LIN {X 0,Y 366.643,Z 618.897,A -85,B 0,C 180,E1 13820.841,E2 13820.841} C_VEL
LIN {X 0,Y 360.03,Z 667.651,A -85,B 0,C 180,E1 13819.206,E2 13819.206} C_VEL
LIN {X 0,Y 355.595,Z 700.826,A -85,B 0,C 180,E1 13817.811,E2 13817.811} C_VEL
LIN {X 0,Y 351.844,Z 722.205,A -85,B 0,C 180,E1 13816.612,E2 13816.612} C_VEL
LIN {X 0,Y 347.315,Z 742.561,A -85,B 0,C 180,E1 13815.174,E2 13815.174} C_VEL
LIN {X 0,Y 342.182,Z 761.879,A -85,B 0,C 180,E1 13813.484,E2 13813.484} C_VEL
LIN {X 0,Y 336.449,Z 780.451,A -85,B 0,C 180,E1 13811.503,E2 13811.503} C_VEL
LIN {X 0,Y 330.364,Z 797.932,A -85,B 0,C 180,E1 13809.24,E2 13809.24} C_VEL
LIN {X 0,Y 324.065,Z 814.382,A -85,B 0,C 180,E1 13806.657,E2 13806.657} C_VEL
LIN {X 0,Y 317.926,Z 829.258,A -85,B 0,C 180,E1 13803.826,E2 13803.826} C_VEL
LIN {X 0,Y 311.925,Z 843.014,A -85,B 0,C 180,E1 13800.643,E2 13800.643} C_VEL
LIN {X 0,Y 306.423,Z 855.219,A -85,B 0,C 180,E1 13797.183,E2 13797.183} C_VEL
LIN {X 0,Y 301.577,Z 865.858,A -85,B 0,C 180,E1 13793.445,E2 13793.445} C_VEL
LIN {X 0,Y 297.526,Z 874.902,A -85,B 0,C 180,E1 13789.433,E2 13789.433} C_VEL
LIN {X 0,Y 294.517,Z 881.994,A -85,B 0,C 180,E1 13785.356,E2 13785.356} C_VEL
LIN {X 0,Y 292.358,Z 887.482,A -85,B 0,C 180,E1 13781.042,E2 13781.042} C_VEL
LIN {X 0,Y 291.105,Z 891.11,A -85,B 0,C 180,E1 13776.707,E2 13776.707} C_VEL
LIN {X 0,Y 290.551,Z 892.885,A -85,B 0,C 180,E1 13772.564,E2 13772.564} C_VEL
LIN {X 0,Y 290.477,Z 893.097,A -85,B 0,C 180,E1 13768.619,E2 13768.619} C_VEL
LIN {X 0,Y 290.873,Z 891.794,A -85,B 0,C 180,E1 13764.477,E2 13764.477} C_VEL
LIN {X 0,Y 291.835,Z 888.902,A -85,B 0,C 180,E1 13760.335,E2 13760.335} C_VEL
LIN {X 0,Y 293.569,Z 884.354,A -85,B 0,C 180,E1 13756.207,E2 13756.207} C_VEL
LIN {X 0,Y 296.202,Z 878.044,A -85,B 0,C 180,E1 13752.11,E2 13752.11} C_VEL
LIN {X 0,Y 299.836,Z 869.83,A -85,B 0,C 180,E1 13748.069,E2 13748.069} C_VEL
LIN {X 0,Y 304.281,Z 860.081,A -85,B 0,C 180,E1 13744.294,E2 13744.294} C_VEL
LIN {X 0,Y 309.693,Z 848.18,A -85,B 0,C 180,E1 13740.61,E2 13740.61} C_VEL
LIN {X 0,Y 315.388,Z 835.383,A -85,B 0,C 180,E1 13737.387,E2 13737.387} C_VEL
LIN {X 0,Y 321.456,Z 821.111,A -85,B 0,C 180,E1 13734.432,E2 13734.432} C_VEL
LIN {X 0,Y 327.943,Z 804.743,A -85,B 0,C 180,E1 13731.65,E2 13731.65} C_VEL
LIN {X 0,Y 334.1,Z 787.79,A -85,B 0,C 180,E1 13729.275,E2 13729.275} C_VEL
LIN {X 0,Y 339.952,Z 769.852,A -85,B 0,C 180,E1 13727.201,E2 13727.201} C_VEL
LIN {X 0,Y 341.959,Z 763.048,A -85,B 0,C 180,E1 13726.517,E2 13726.517} C_VEL
LIN {X 0,Y 343.111,Z 756.729,A -85,B 0,C 180,E1 13725.787,E2 13725.787} C_VEL
LIN {X 0,Y 343.287,Z 740.949,A -85,B 0,C 180,E1 13723.705,E2 13723.705} C_VEL
LIN {X 0,Y 344.169,Z 734.277,A -85,B 0,C 180,E1 13723.068,E2 13723.068} C_VEL
LIN {X 0,Y 348.496,Z 713.392,A -85,B 0,C 180,E1 13721.732,E2 13721.732} C_VEL
LIN {X 0,Y 351.931,Z 691.641,A -85,B 0,C 180,E1 13720.649,E2 13720.649} C_VEL
LIN {X 0,Y 357.689,Z 649.532,A -85,B 0,C 180,E1 13719.026,E2 13719.026} C_VEL
LIN {X 0,Y 364.593,Z 600.879,A -85,B 0,C 180,E1 13717.565,E2 13717.565} C_VEL
LIN {X 0,Y 370.767,Z 550.378,A -85,B 0,C 180,E1 13716.308,E2 13716.308} C_VEL
LIN {X 0,Y 375.514,Z 499.907,A -85,B 0,C 180,E1 13715.262,E2 13715.262} C_VEL
LIN {X 0,Y 380.163,Z 439.411,A -85,B 0,C 180,E1 13714.164,E2 13714.164} C_VEL
LIN {X 0,Y 386.666,Z 411.148,A -85,B 0,C 180,E1 13713.223,E2 13713.223} C_VEL
LIN {X 0,Y 381.926,Z 396.352,A -85,B 0,C 180,E1 13710.437,E2 13710.437} C_VEL
LIN {X 0,Y 376.863,Z 382.161,A -85,B 0,C 180,E1 13707.323,E2 13707.323} C_VEL
LIN {X 0,Y 372.149,Z 370.419,A -85,B 0,C 180,E1 13704.273,E2 13704.273} C_VEL
LIN {X 0,Y 367.922,Z 360.719,A -85,B 0,C 180,E1 13701.315,E2 13701.315} C_VEL
LIN {X 0,Y 364.04,Z 352.331,A -85,B 0,C 180,E1 13698.247,E2 13698.247} C_VEL
LIN {X 0,Y 361.674,Z 347.588,A -85,B 0,C 180,E1 13696.214,E2 13696.214} C_VEL
LIN {X 0,Y 359.895,Z 343.923,A -85,B 0,C 180,E1 13694.48,E2 13694.48} C_VEL
LIN {X 0,Y 357.988,Z 339.875,A -85,B 0,C 180,E1 13692.256,E2 13692.256} C_VEL
LIN {X 0,Y 355.585,Z 335.237,A -85,B 0,C 180,E1 13689.223,E2 13689.223} C_VEL
LIN {X 0,Y 353.736,Z 331.636,A -85,B 0,C 180,E1 13685.841,E2 13685.841} C_VEL
LIN {X 0,Y 353.406,Z 330.304,A -85,B 0,C 180,E1 13684.706,E2 13684.706} C_VEL
LIN {X 0,Y 352.685,Z 328.775,A -85,B 0,C 180,E1 13678.375,E2 13678.375} C_VEL
LIN {X 0,Y 354.065,Z 329.807,A -85,B 0,C 180,E1 13673.677,E2 13673.677} C_VEL
LIN {X 0,Y 355.236,Z 330.811,A -85,B 0,C 180,E1 13671.828,E2 13671.828} C_VEL
LIN {X 0,Y 356.963,Z 342.871,A -85,B 0,C 180,E1 13667.626,E2 13667.626} C_VEL
LIN {X 0,Y 360.086,Z 356.086,A -85,B 0,C 180,E1 13663.671,E2 13663.671} C_VEL
LIN {X 0,Y 366.35,Z 375.856,A -85,B 0,C 180,E1 13658.715,E2 13658.715} C_VEL
LIN {X 0,Y 369.886,Z 385.971,A -85,B 0,C 180,E1 13656.543,E2 13656.543} C_VEL
LIN {X 0,Y 376.95,Z 407.665,A -85,B 0,C 180,E1 13652.729,E2 13652.729} C_VEL
LIN {X 0,Y 356.204,Z 579.083,A -85,B 0,C 180,E1 13648.165,E2 13648.165} C_VEL
LIN {X 0,Y 351.392,Z 648.87,A -85,B 0,C 180,E1 13646.675,E2 13646.675} C_VEL
LIN {X 0,Y 347.833,Z 683.011,A -85,B 0,C 180,E1 13645.721,E2 13645.721} C_VEL
LIN {X 0,Y 343.149,Z 716.181,A -85,B 0,C 180,E1 13644.541,E2 13644.541} C_VEL
LIN {X 0,Y 338.014,Z 746.973,A -85,B 0,C 180,E1 13643.133,E2 13643.133} C_VEL
LIN {X 0,Y 332.497,Z 776.814,A -85,B 0,C 180,E1 13641.433,E2 13641.433} C_VEL
LIN {X 0,Y 326.517,Z 805.796,A -85,B 0,C 180,E1 13639.415,E2 13639.415} C_VEL
LIN {X 0,Y 322.047,Z 824.838,A -85,B 0,C 180,E1 13637.773,E2 13637.773} C_VEL
LIN {X 0,Y 316.988,Z 843.135,A -85,B 0,C 180,E1 13635.845,E2 13635.845} C_VEL
LIN {X 0,Y 311.435,Z 861.14,A -85,B 0,C 180,E1 13633.525,E2 13633.525} C_VEL
LIN {X 0,Y 305.778,Z 878.186,A -85,B 0,C 180,E1 13630.844,E2 13630.844} C_VEL
LIN {X 0,Y 300.361,Z 893.477,A -85,B 0,C 180,E1 13627.911,E2 13627.911} C_VEL
LIN {X 0,Y 295.216,Z 907.713,A -85,B 0,C 180,E1 13624.61,E2 13624.61} C_VEL
LIN {X 0,Y 290.74,Z 920.364,A -85,B 0,C 180,E1 13621.055,E2 13621.055} C_VEL
LIN {X 0,Y 286.97,Z 931.798,A -85,B 0,C 180,E1 13617.158,E2 13617.158} C_VEL
LIN {X 0,Y 284.132,Z 941.659,A -85,B 0,C 180,E1 13612.993,E2 13612.993} C_VEL
LIN {X 0,Y 282.324,Z 949.983,A -85,B 0,C 180,E1 13608.587,E2 13608.587} C_VEL
LIN {X 0,Y 281.545,Z 956.442,A -85,B 0,C 180,E1 13604.176,E2 13604.176} C_VEL
LIN {X 0,Y 281.547,Z 960.921,A -85,B 0,C 180,E1 13600.021,E2 13600.021} C_VEL
LIN {X 0,Y 282.01,Z 964.446,A -85,B 0,C 180,E1 13595.289,E2 13595.289} C_VEL
LIN {X 0,Y 282.157,Z 966.76,A -85,B 0,C 180,E1 13591.624,E2 13591.624} C_VEL
LIN {X 0,Y 281.994,Z 967.796,A -85,B 0,C 180,E1 13588.171,E2 13588.171} C_VEL
LIN {X 0,Y 281.58,Z 967.758,A -85,B 0,C 180,E1 13584.702,E2 13584.702} C_VEL
LIN {X 0,Y 281.082,Z 966.455,A -85,B 0,C 180,E1 13580.582,E2 13580.582} C_VEL
LIN {X 0,Y 281.08,Z 963.184,A -85,B 0,C 180,E1 13575.581,E2 13575.581} C_VEL
LIN {X 0,Y 282.123,Z 958.691,A -85,B 0,C 180,E1 13570.97,E2 13570.97} C_VEL
LIN {X 0,Y 285.023,Z 951.705,A -85,B 0,C 180,E1 13565.546,E2 13565.546} C_VEL
LIN {X 0,Y 290.041,Z 942.875,A -85,B 0,C 180,E1 13560.236,E2 13560.236} C_VEL
LIN {X 0,Y 297.987,Z 931.43,A -85,B 0,C 180,E1 13554.75,E2 13554.75} C_VEL
LIN {X 0,Y 308.228,Z 918.66,A -85,B 0,C 180,E1 13549.792,E2 13549.792} C_VEL
LIN {X 0,Y 320.962,Z 904.077,A -85,B 0,C 180,E1 13545.246,E2 13545.246} C_VEL
LIN {X 0,Y 336.752,Z 887.173,A -85,B 0,C 180,E1 13541.011,E2 13541.011} C_VEL
LIN {X 0,Y 353.463,Z 870.171,A -85,B 0,C 180,E1 13537.62,E2 13537.62} C_VEL
LIN {X 0,Y 355.449,Z 868.133,A -85,B 0,C 180,E1 13537.244,E2 13537.244} C_VEL
LIN {X 0,Y 339.797,Z 879.829,A -85,B 0,C 180,E1 13534.197,E2 13534.197} C_VEL
LIN {X 0,Y 326.256,Z 889.867,A -85,B 0,C 180,E1 13530.785,E2 13530.785} C_VEL
LIN {X 0,Y 315.116,Z 897.821,A -85,B 0,C 180,E1 13527.189,E2 13527.189} C_VEL
LIN {X 0,Y 306.095,Z 903.73,A -85,B 0,C 180,E1 13523.486,E2 13523.486} C_VEL
LIN {X 0,Y 298.648,Z 907.843,A -85,B 0,C 180,E1 13519.561,E2 13519.561} C_VEL
LIN {X 0,Y 292.968,Z 909.937,A -85,B 0,C 180,E1 13515.642,E2 13515.642} C_VEL
LIN {X 0,Y 288.828,Z 910.181,A -85,B 0,C 180,E1 13511.786,E2 13511.786} C_VEL
LIN {X 0,Y 285.968,Z 908.753,A -85,B 0,C 180,E1 13508.04,E2 13508.04} C_VEL
LIN {X 0,Y 283.949,Z 905.358,A -85,B 0,C 180,E1 13504.039,E2 13504.039} C_VEL
LIN {X 0,Y 282.868,Z 900.293,A -85,B 0,C 180,E1 13500.203,E2 13500.203} C_VEL
LIN {X 0,Y 282.437,Z 893.734,A -85,B 0,C 180,E1 13496.55,E2 13496.55} C_VEL
LIN {X 0,Y 282.553,Z 885.362,A -85,B 0,C 180,E1 13492.885,E2 13492.885} C_VEL
LIN {X 0,Y 283.163,Z 875.563,A -85,B 0,C 180,E1 13489.419,E2 13489.419} C_VEL
LIN {X 0,Y 284.429,Z 862.976,A -85,B 0,C 180,E1 13485.754,E2 13485.754} C_VEL
LIN {X 0,Y 286.155,Z 849.601,A -85,B 0,C 180,E1 13482.512,E2 13482.512} C_VEL
LIN {X 0,Y 288.324,Z 834.796,A -85,B 0,C 180,E1 13479.496,E2 13479.496} C_VEL
LIN {X 0,Y 290.976,Z 818.009,A -85,B 0,C 180,E1 13476.605,E2 13476.605} C_VEL
LIN {X 0,Y 293.944,Z 799.899,A -85,B 0,C 180,E1 13473.972,E2 13473.972} C_VEL
LIN {X 0,Y 297.289,Z 779.355,A -85,B 0,C 180,E1 13471.471,E2 13471.471} C_VEL
LIN {X 0,Y 300.696,Z 757.667,A -85,B 0,C 180,E1 13469.308,E2 13469.308} C_VEL
LIN {X 0,Y 304.018,Z 734.908,A -85,B 0,C 180,E1 13467.47,E2 13467.47} C_VEL
LIN {X 0,Y 304.579,Z 731.096,A -85,B 0,C 180,E1 13467.184,E2 13467.184} C_VEL
LIN {X 0,Y 306.11,Z 730.891,A -85,B 0,C 180,E1 13466.718,E2 13466.718} C_VEL
LIN {X 0,Y 308.996,Z 728.323,A -85,B 0,C 180,E1 13466.18,E2 13466.18} C_VEL
LIN {X 0,Y 313.01,Z 722.831,A -85,B 0,C 180,E1 13465.68,E2 13465.68} C_VEL
LIN {X 0,Y 315.541,Z 718.67,A -85,B 0,C 180,E1 13465.443,E2 13465.443} C_VEL
LIN {X 0,Y 319.129,Z 715.537,A -85,B 0,C 180,E1 13464.795,E2 13464.795} C_VEL
LIN {X 0,Y 323.29,Z 709.874,A -85,B 0,C 180,E1 13464.256,E2 13464.256} C_VEL
LIN {X 0,Y 328.312,Z 700.656,A -85,B 0,C 180,E1 13463.823,E2 13463.823} C_VEL
LIN {X 0,Y 329.111,Z 699.455,A -85,B 0,C 180,E1 13463.723,E2 13463.723} C_VEL
LIN {X 0,Y 333.176,Z 694.404,A -85,B 0,C 180,E1 13463.141,E2 13463.141} C_VEL
LIN {X 0,Y 337.92,Z 686.155,A -85,B 0,C 180,E1 13462.657,E2 13462.657} C_VEL
LIN {X 0,Y 342.453,Z 676.446,A -85,B 0,C 180,E1 13462.34,E2 13462.34} C_VEL
LIN {X 0,Y 347.169,Z 669.599,A -85,B 0,C 180,E1 13461.766,E2 13461.766} C_VEL
LIN {X 0,Y 352.346,Z 659.543,A -85,B 0,C 180,E1 13461.329,E2 13461.329} C_VEL
LIN {X 0,Y 355.868,Z 651.493,A -85,B 0,C 180,E1 13461.105,E2 13461.105} C_VEL
LIN {X 0,Y 357.637,Z 649.135,A -85,B 0,C 180,E1 13460.884,E2 13460.884} C_VEL
LIN {X 0,Y 351.863,Z 690.96,A -85,B 0,C 180,E1 13459.267,E2 13459.267} C_VEL
LIN {X 0,Y 348.458,Z 712.778,A -85,B 0,C 180,E1 13458.189,E2 13458.189} C_VEL
LIN {X 0,Y 344.081,Z 734.017,A -85,B 0,C 180,E1 13456.836,E2 13456.836} C_VEL
LIN {X 0,Y 339.136,Z 753.596,A -85,B 0,C 180,E1 13455.28,E2 13455.28} C_VEL
LIN {X 0,Y 333.354,Z 772.976,A -85,B 0,C 180,E1 13453.384,E2 13453.384} C_VEL
LIN {X 0,Y 327.127,Z 791.223,A -85,B 0,C 180,E1 13451.2,E2 13451.2} C_VEL
LIN {X 0,Y 320.606,Z 808.342,A -85,B 0,C 180,E1 13448.705,E2 13448.705} C_VEL
LIN {X 0,Y 314.356,Z 823.41,A -85,B 0,C 180,E1 13446.047,E2 13446.047} C_VEL
LIN {X 0,Y 308.117,Z 837.495,A -85,B 0,C 180,E1 13443.038,E2 13443.038} C_VEL
LIN {X 0,Y 302.257,Z 850.138,A -85,B 0,C 180,E1 13439.75,E2 13439.75} C_VEL
LIN {X 0,Y 296.681,Z 861.846,A -85,B 0,C 180,E1 13435.985,E2 13435.985} C_VEL
LIN {X 0,Y 292.104,Z 871.467,A -85,B 0,C 180,E1 13432.12,E2 13432.12} C_VEL
LIN {X 0,Y 288.361,Z 879.551,A -85,B 0,C 180,E1 13427.975,E2 13427.975} C_VEL
LIN {X 0,Y 285.658,Z 885.743,A -85,B 0,C 180,E1 13423.77,E2 13423.77} C_VEL
LIN {X 0,Y 283.884,Z 890.175,A -85,B 0,C 180,E1 13419.524,E2 13419.524} C_VEL
LIN {X 0,Y 282.942,Z 892.841,A -85,B 0,C 180,E1 13415.475,E2 13415.475} C_VEL
LIN {X 0,Y 282.536,Z 894.107,A -85,B 0,C 180,E1 13411.217,E2 13411.217} C_VEL
LIN {X 0,Y 282.626,Z 893.861,A -85,B 0,C 180,E1 13407.161,E2 13407.161} C_VEL
LIN {X 0,Y 283.235,Z 892.063,A -85,B 0,C 180,E1 13402.903,E2 13402.903} C_VEL
LIN {X 0,Y 284.594,Z 888.422,A -85,B 0,C 180,E1 13398.448,E2 13398.448} C_VEL
LIN {X 0,Y 286.916,Z 882.914,A -85,B 0,C 180,E1 13394.02,E2 13394.02} C_VEL
LIN {X 0,Y 290.121,Z 875.798,A -85,B 0,C 180,E1 13389.84,E2 13389.84} C_VEL
LIN {X 0,Y 294.418,Z 866.728,A -85,B 0,C 180,E1 13385.736,E2 13385.736} C_VEL
LIN {X 0,Y 299.529,Z 856.058,A -85,B 0,C 180,E1 13381.921,E2 13381.921} C_VEL
LIN {X 0,Y 305.402,Z 843.624,A -85,B 0,C 180,E1 13378.348,E2 13378.348} C_VEL
LIN {X 0,Y 311.589,Z 830.016,A -85,B 0,C 180,E1 13375.166,E2 13375.166} C_VEL
LIN {X 0,Y 318.201,Z 814.584,A -85,B 0,C 180,E1 13372.211,E2 13372.211} C_VEL
LIN {X 0,Y 324.768,Z 797.965,A -85,B 0,C 180,E1 13369.603,E2 13369.603} C_VEL
LIN {X 0,Y 331.11,Z 780.235,A -85,B 0,C 180,E1 13367.317,E2 13367.317} C_VEL
LIN {X 0,Y 336.784,Z 762.36,A -85,B 0,C 180,E1 13365.412,E2 13365.412} C_VEL
LIN {X 0,Y 342.19,Z 742.493,A -85,B 0,C 180,E1 13363.681,E2 13363.681} C_VEL
LIN {X 0,Y 344.169,Z 734.277,A -85,B 0,C 180,E1 13363.068,E2 13363.068} C_VEL
LIN {X 0,Y 345.161,Z 727.504,A -85,B 0,C 180,E1 13362.456,E2 13362.456} C_VEL
LIN {X 0,Y 344.675,Z 710.571,A -85,B 0,C 180,E1 13360.65,E2 13360.65} C_VEL
LIN {X 0,Y 345.144,Z 703.415,A -85,B 0,C 180,E1 13360.16,E2 13360.16} C_VEL
LIN {X 0,Y 350.733,Z 664.574,A -85,B 0,C 180,E1 13358.521,E2 13358.521} C_VEL
LIN {X 0,Y 356.943,Z 622.303,A -85,B 0,C 180,E1 13357.123,E2 13357.123} C_VEL
LIN {X 0,Y 363.707,Z 572.194,A -85,B 0,C 180,E1 13355.791,E2 13355.791} C_VEL
LIN {X 0,Y 369.148,Z 521.87,A -85,B 0,C 180,E1 13354.67,E2 13354.67} C_VEL
LIN {X 0,Y 374.356,Z 456.234,A -85,B 0,C 180,E1 13353.457,E2 13353.457} C_VEL
LIN {X 0,Y 375.644,Z 442.026,A -85,B 0,C 180,E1 13353.187,E2 13353.187} C_VEL
LIN {X 0,Y 381.952,Z 414.888,A -85,B 0,C 180,E1 13352.305,E2 13352.305} C_VEL
LIN {X 0,Y 377.182,Z 399.775,A -85,B 0,C 180,E1 13349.369,E2 13349.369} C_VEL
LIN {X 0,Y 372.444,Z 386.352,A -85,B 0,C 180,E1 13346.294,E2 13346.294} C_VEL
LIN {X 0,Y 367.993,Z 374.96,A -85,B 0,C 180,E1 13343.203,E2 13343.203} C_VEL
LIN {X 0,Y 363.588,Z 364.648,A -85,B 0,C 180,E1 13339.897,E2 13339.897} C_VEL
LIN {X 0,Y 359.792,Z 356.235,A -85,B 0,C 180,E1 13336.55,E2 13336.55} C_VEL
LIN {X 0,Y 357.363,Z 351.267,A -85,B 0,C 180,E1 13334.171,E2 13334.171} C_VEL
LIN {X 0,Y 355.676,Z 347.381,A -85,B 0,C 180,E1 13332.007,E2 13332.007} C_VEL
LIN {X 0,Y 353.511,Z 342.934,A -85,B 0,C 180,E1 13329.114,E2 13329.114} C_VEL
LIN {X 0,Y 351.685,Z 339.321,A -85,B 0,C 180,E1 13325.675,E2 13325.675} C_VEL
LIN {X 0,Y 351.434,Z 338.035,A -85,B 0,C 180,E1 13324.569,E2 13324.569} C_VEL
LIN {X 0,Y 350.792,Z 336.546,A -85,B 0,C 180,E1 13318.203,E2 13318.203} C_VEL
LIN {X 0,Y 352.569,Z 337.811,A -85,B 0,C 180,E1 13313.159,E2 13313.159} C_VEL
LIN {X 0,Y 353.238,Z 338.552,A -85,B 0,C 180,E1 13312.068,E2 13312.068} C_VEL
LIN {X 0,Y 354.771,Z 350.186,A -85,B 0,C 180,E1 13308.044,E2 13308.044} C_VEL
LIN {X 0,Y 357.683,Z 362.885,A -85,B 0,C 180,E1 13304.225,E2 13304.225} C_VEL
LIN {X 0,Y 363.605,Z 382.359,A -85,B 0,C 180,E1 13299.307,E2 13299.307} C_VEL
LIN {X 0,Y 366.869,Z 392.296,A -85,B 0,C 180,E1 13297.146,E2 13297.146} C_VEL
LIN {X 0,Y 372.922,Z 411.537,A -85,B 0,C 180,E1 13293.732,E2 13293.732} C_VEL
LIN {X 0,Y 351.644,Z 581.817,A -85,B 0,C 180,E1 13289.192,E2 13289.192} C_VEL
LIN {X 0,Y 347.333,Z 643.921,A -85,B 0,C 180,E1 13287.885,E2 13287.885} C_VEL
LIN {X 0,Y 343.821,Z 677.097,A -85,B 0,C 180,E1 13286.978,E2 13286.978} C_VEL
LIN {X 0,Y 339.246,Z 709.541,A -85,B 0,C 180,E1 13285.859,E2 13285.859} C_VEL
LIN {X 0,Y 334.198,Z 739.62,A -85,B 0,C 180,E1 13284.561,E2 13284.561} C_VEL
LIN {X 0,Y 329.139,Z 766.452,A -85,B 0,C 180,E1 13283.092,E2 13283.092} C_VEL
LIN {X 0,Y 323.665,Z 792.898,A -85,B 0,C 180,E1 13281.388,E2 13281.388} C_VEL
LIN {X 0,Y 318.9,Z 813.963,A -85,B 0,C 180,E1 13279.767,E2 13279.767} C_VEL
LIN {X 0,Y 313.811,Z 833.029,A -85,B 0,C 180,E1 13277.936,E2 13277.936} C_VEL
LIN {X 0,Y 308.277,Z 851.263,A -85,B 0,C 180,E1 13275.785,E2 13275.785} C_VEL
LIN {X 0,Y 302.587,Z 868.119,A -85,B 0,C 180,E1 13273.366,E2 13273.366} C_VEL
LIN {X 0,Y 296.762,Z 884.18,A -85,B 0,C 180,E1 13270.563,E2 13270.563} C_VEL
LIN {X 0,Y 291.203,Z 898.921,A -85,B 0,C 180,E1 13267.427,E2 13267.427} C_VEL
LIN {X 0,Y 285.848,Z 912.994,A -85,B 0,C 180,E1 13263.792,E2 13263.792} C_VEL
LIN {X 0,Y 281.5,Z 924.876,A -85,B 0,C 180,E1 13260.055,E2 13260.055} C_VEL
LIN {X 0,Y 277.904,Z 935.632,A -85,B 0,C 180,E1 13255.908,E2 13255.908} C_VEL
LIN {X 0,Y 275.364,Z 944.751,A -85,B 0,C 180,E1 13251.515,E2 13251.515} C_VEL
LIN {X 0,Y 273.934,Z 952.193,A -85,B 0,C 180,E1 13246.978,E2 13246.978} C_VEL
LIN {X 0,Y 273.513,Z 957.825,A -85,B 0,C 180,E1 13242.456,E2 13242.456} C_VEL
LIN {X 0,Y 273.762,Z 961.703,A -85,B 0,C 180,E1 13237.978,E2 13237.978} C_VEL
LIN {X 0,Y 274.215,Z 964.141,A -85,B 0,C 180,E1 13233.763,E2 13233.763} C_VEL
LIN {X 0,Y 274.249,Z 965.886,A -85,B 0,C 180,E1 13230.418,E2 13230.418} C_VEL
LIN {X 0,Y 273.977,Z 966.635,A -85,B 0,C 180,E1 13227.071,E2 13227.071} C_VEL
LIN {X 0,Y 273.434,Z 966.354,A -85,B 0,C 180,E1 13223.28,E2 13223.28} C_VEL
LIN {X 0,Y 272.998,Z 964.568,A -85,B 0,C 180,E1 13218.593,E2 13218.593} C_VEL
LIN {X 0,Y 273.392,Z 961.021,A -85,B 0,C 180,E1 13213.643,E2 13213.643} C_VEL
LIN {X 0,Y 275.26,Z 955.619,A -85,B 0,C 180,E1 13208.252,E2 13208.252} C_VEL
LIN {X 0,Y 279.247,Z 948.099,A -85,B 0,C 180,E1 13202.721,E2 13202.721} C_VEL
LIN {X 0,Y 286.111,Z 938.203,A -85,B 0,C 180,E1 13196.963,E2 13196.963} C_VEL
LIN {X 0,Y 295.749,Z 926.427,A -85,B 0,C 180,E1 13191.532,E2 13191.532} C_VEL
LIN {X 0,Y 308.63,Z 912.329,A -85,B 0,C 180,E1 13186.364,E2 13186.364} C_VEL
LIN {X 0,Y 324.964,Z 895.932,A -85,B 0,C 180,E1 13181.609,E2 13181.609} C_VEL
LIN {X 0,Y 342.561,Z 879.263,A -85,B 0,C 180,E1 13177.804,E2 13177.804} C_VEL
LIN {X 0,Y 345.779,Z 876.2,A -85,B 0,C 180,E1 13177.183,E2 13177.183} C_VEL
LIN {X 0,Y 329.727,Z 887.067,A -85,B 0,C 180,E1 13173.916,E2 13173.916} C_VEL
LIN {X 0,Y 316.341,Z 895.907,A -85,B 0,C 180,E1 13170.38,E2 13170.38} C_VEL
LIN {X 0,Y 305.348,Z 902.734,A -85,B 0,C 180,E1 13166.655,E2 13166.655} C_VEL
LIN {X 0,Y 296.124,Z 907.761,A -85,B 0,C 180,E1 13162.64,E2 13162.64} C_VEL
LIN {X 0,Y 288.937,Z 910.728,A -85,B 0,C 180,E1 13158.565,E2 13158.565} C_VEL
LIN {X 0,Y 283.548,Z 911.729,A -85,B 0,C 180,E1 13154.5,E2 13154.5} C_VEL
LIN {X 0,Y 279.712,Z 910.927,A -85,B 0,C 180,E1 13150.504,E2 13150.504} C_VEL
LIN {X 0,Y 277.138,Z 908.494,A -85,B 0,C 180,E1 13146.63,E2 13146.63} C_VEL
LIN {X 0,Y 275.432,Z 904.039,A -85,B 0,C 180,E1 13142.497,E2 13142.497} C_VEL
LIN {X 0,Y 274.615,Z 897.929,A -85,B 0,C 180,E1 13138.539,E2 13138.539} C_VEL
LIN {X 0,Y 274.433,Z 890.313,A -85,B 0,C 180,E1 13134.774,E2 13134.774} C_VEL
LIN {X 0,Y 274.82,Z 880.793,A -85,B 0,C 180,E1 13130.999,E2 13130.999} C_VEL
LIN {X 0,Y 275.674,Z 870.498,A -85,B 0,C 180,E1 13127.643,E2 13127.643} C_VEL
LIN {X 0,Y 277.198,Z 857.439,A -85,B 0,C 180,E1 13124.089,E2 13124.089} C_VEL
LIN {X 0,Y 279.257,Z 842.882,A -85,B 0,C 180,E1 13120.767,E2 13120.767} C_VEL
LIN {X 0,Y 281.877,Z 826.293,A -85,B 0,C 180,E1 13117.584,E2 13117.584} C_VEL
LIN {X 0,Y 284.925,Z 807.951,A -85,B 0,C 180,E1 13114.651,E2 13114.651} C_VEL
LIN {X 0,Y 288.304,Z 787.762,A -85,B 0,C 180,E1 13111.97,E2 13111.97} C_VEL
LIN {X 0,Y 291.752,Z 766.54,A -85,B 0,C 180,E1 13109.635,E2 13109.635} C_VEL
LIN {X 0,Y 294.859,Z 747.2,A -85,B 0,C 180,E1 13107.832,E2 13107.832} C_VEL
LIN {X 0,Y 296.39,Z 747.01,A -85,B 0,C 180,E1 13107.332,E2 13107.332} C_VEL
LIN {X 0,Y 299.207,Z 744.812,A -85,B 0,C 180,E1 13106.766,E2 13106.766} C_VEL
LIN {X 0,Y 303.035,Z 740.398,A -85,B 0,C 180,E1 13106.253,E2 13106.253} C_VEL
LIN {X 0,Y 304.712,Z 738.085,A -85,B 0,C 180,E1 13106.093,E2 13106.093} C_VEL
LIN {X 0,Y 308.153,Z 735.594,A -85,B 0,C 180,E1 13105.4,E2 13105.4} C_VEL
LIN {X 0,Y 312.287,Z 731.048,A -85,B 0,C 180,E1 13104.807,E2 13104.807} C_VEL
LIN {X 0,Y 317.192,Z 724.171,A -85,B 0,C 180,E1 13104.325,E2 13104.325} C_VEL
LIN {X 0,Y 321.621,Z 719.801,A -85,B 0,C 180,E1 13103.63,E2 13103.63} C_VEL
LIN {X 0,Y 326.394,Z 713.32,A -85,B 0,C 180,E1 13103.099,E2 13103.099} C_VEL
LIN {X 0,Y 331.706,Z 704.206,A -85,B 0,C 180,E1 13102.652,E2 13102.652} C_VEL
LIN {X 0,Y 336.52,Z 698.024,A -85,B 0,C 180,E1 13102.044,E2 13102.044} C_VEL
LIN {X 0,Y 341.759,Z 688.852,A -85,B 0,C 180,E1 13101.558,E2 13101.558} C_VEL
LIN {X 0,Y 345.773,Z 680.521,A -85,B 0,C 180,E1 13101.292,E2 13101.292} C_VEL
LIN {X 0,Y 348.925,Z 676.153,A -85,B 0,C 180,E1 13100.917,E2 13100.917} C_VEL
LIN {X 0,Y 344.608,Z 705.687,A -85,B 0,C 180,E1 13099.61,E2 13099.61} C_VEL
LIN {X 0,Y 340.76,Z 725.9,A -85,B 0,C 180,E1 13098.439,E2 13098.439} C_VEL
LIN {X 0,Y 335.873,Z 746.278,A -85,B 0,C 180,E1 13096.958,E2 13096.958} C_VEL
LIN {X 0,Y 330.387,Z 765.45,A -85,B 0,C 180,E1 13095.231,E2 13095.231} C_VEL
LIN {X 0,Y 324.254,Z 783.887,A -85,B 0,C 180,E1 13093.202,E2 13093.202} C_VEL
LIN {X 0,Y 317.754,Z 801.203,A -85,B 0,C 180,E1 13090.884,E2 13090.884} C_VEL
LIN {X 0,Y 311.233,Z 817.009,A -85,B 0,C 180,E1 13088.32,E2 13088.32} C_VEL
LIN {X 0,Y 304.434,Z 832.212,A -85,B 0,C 180,E1 13085.314,E2 13085.314} C_VEL
LIN {X 0,Y 297.971,Z 845.825,A -85,B 0,C 180,E1 13082.019,E2 13082.019} C_VEL
LIN {X 0,Y 292.018,Z 857.892,A -85,B 0,C 180,E1 13078.421,E2 13078.421} C_VEL
LIN {X 0,Y 286.751,Z 868.407,A -85,B 0,C 180,E1 13074.516,E2 13074.516} C_VEL
LIN {X 0,Y 282.514,Z 876.971,A -85,B 0,C 180,E1 13070.511,E2 13070.511} C_VEL
LIN {X 0,Y 279.162,Z 884.043,A -85,B 0,C 180,E1 13066.223,E2 13066.223} C_VEL
LIN {X 0,Y 276.738,Z 889.511,A -85,B 0,C 180,E1 13061.674,E2 13061.674} C_VEL
LIN {X 0,Y 275.316,Z 893.121,A -85,B 0,C 180,E1 13057.093,E2 13057.093} C_VEL
LIN {X 0,Y 274.688,Z 894.887,A -85,B 0,C 180,E1 13052.712,E2 13052.712} C_VEL
LIN {X 0,Y 274.606,Z 895.099,A -85,B 0,C 180,E1 13048.54,E2 13048.54} C_VEL
LIN {X 0,Y 275.057,Z 893.802,A -85,B 0,C 180,E1 13044.158,E2 13044.158} C_VEL
LIN {X 0,Y 276.147,Z 890.921,A -85,B 0,C 180,E1 13039.78,E2 13039.78} C_VEL
LIN {X 0,Y 278.099,Z 886.385,A -85,B 0,C 180,E1 13035.423,E2 13035.423} C_VEL
LIN {X 0,Y 280.98,Z 880.228,A -85,B 0,C 180,E1 13031.189,E2 13031.189} C_VEL
LIN {X 0,Y 284.857,Z 872.344,A -85,B 0,C 180,E1 13027.069,E2 13027.069} C_VEL
LIN {X 0,Y 289.699,Z 862.703,A -85,B 0,C 180,E1 13023.119,E2 13023.119} C_VEL
LIN {X 0,Y 295.568,Z 850.942,A -85,B 0,C 180,E1 13019.281,E2 13019.281} C_VEL
LIN {X 0,Y 301.712,Z 838.27,A -85,B 0,C 180,E1 13015.939,E2 13015.939} C_VEL
LIN {X 0,Y 308.232,Z 824.136,A -85,B 0,C 180,E1 13012.888,E2 13012.888} C_VEL
LIN {X 0,Y 315.125,Z 808.088,A -85,B 0,C 180,E1 13010.05,E2 13010.05} C_VEL
LIN {X 0,Y 321.753,Z 791.181,A -85,B 0,C 180,E1 13007.596,E2 13007.596} C_VEL
LIN {X 0,Y 327.984,Z 773.454,A -85,B 0,C 180,E1 13005.479,E2 13005.479} C_VEL
LIN {X 0,Y 333.963,Z 753.88,A -85,B 0,C 180,E1 13003.569,E2 13003.569} C_VEL
LIN {X 0,Y 339.078,Z 734.096,A -85,B 0,C 180,E1 13002.003,E2 13002.003} C_VEL
LIN {X 0,Y 343.327,Z 713.93,A -85,B 0,C 180,E1 13000.721,E2 13000.721} C_VEL
LIN {X 0,Y 345.144,Z 703.415,A -85,B 0,C 180,E1 13000.16,E2 13000.16} C_VEL
LIN {X 0,Y 345.652,Z 696.184,A -85,B 0,C 180,E1 12999.693,E2 12999.693} C_VEL
LIN {X 0,Y 344.547,Z 678.435,A -85,B 0,C 180,E1 12998.131,E2 12998.131} C_VEL
LIN {X 0,Y 345.016,Z 671.14,A -85,B 0,C 180,E1 12997.707,E2 12997.707} C_VEL
LIN {X 0,Y 351.317,Z 629.328,A -85,B 0,C 180,E1 12996.269,E2 12996.269} C_VEL
LIN {X 0,Y 358.541,Z 578.262,A -85,B 0,C 180,E1 12994.878,E2 12994.878} C_VEL
LIN {X 0,Y 364.196,Z 528.171,A -85,B 0,C 180,E1 12993.748,E2 12993.748} C_VEL
LIN {X 0,Y 369.295,Z 466.763,A -85,B 0,C 180,E1 12992.597,E2 12992.597} C_VEL
LIN {X 0,Y 371.189,Z 444.83,A -85,B 0,C 180,E1 12992.193,E2 12992.193} C_VEL
LIN {X 0,Y 377.281,Z 418.51,A -85,B 0,C 180,E1 12991.34,E2 12991.34} C_VEL
LIN {X 0,Y 372.706,Z 403.689,A -85,B 0,C 180,E1 12988.35,E2 12988.35} C_VEL
LIN {X 0,Y 368.179,Z 390.746,A -85,B 0,C 180,E1 12985.277,E2 12985.277} C_VEL
LIN {X 0,Y 364.132,Z 380.11,A -85,B 0,C 180,E1 12982.268,E2 12982.268} C_VEL
LIN {X 0,Y 360.372,Z 371.096,A -85,B 0,C 180,E1 12979.28,E2 12979.28} C_VEL
LIN {X 0,Y 357.05,Z 363.402,A -85,B 0,C 180,E1 12976.179,E2 12976.179} C_VEL
LIN {X 0,Y 354.771,Z 358.473,A -85,B 0,C 180,E1 12973.778,E2 12973.778} C_VEL
LIN {X 0,Y 353.222,Z 354.758,A -85,B 0,C 180,E1 12971.677,E2 12971.677} C_VEL
LIN {X 0,Y 351.316,Z 350.5,A -85,B 0,C 180,E1 12968.841,E2 12968.841} C_VEL
LIN {X 0,Y 349.637,Z 346.785,A -85,B 0,C 180,E1 12965.333,E2 12965.333} C_VEL
LIN {X 0,Y 349.523,Z 345.779,A -85,B 0,C 180,E1 12964.43,E2 12964.43} C_VEL
LIN {X 0,Y 348.875,Z 344.313,A -85,B 0,C 180,E1 12958.193,E2 12958.193} C_VEL
LIN {X 0,Y 350.785,Z 345.628,A -85,B 0,C 180,E1 12953.124,E2 12953.124} C_VEL
LIN {X 0,Y 351.232,Z 346.212,A -85,B 0,C 180,E1 12952.352,E2 12952.352} C_VEL
LIN {X 0,Y 352.621,Z 357.497,A -85,B 0,C 180,E1 12948.468,E2 12948.468} C_VEL
LIN {X 0,Y 355.325,Z 369.691,A -85,B 0,C 180,E1 12944.787,E2 12944.787} C_VEL
LIN {X 0,Y 360.791,Z 388.654,A -85,B 0,C 180,E1 12939.95,E2 12939.95} C_VEL
LIN {X 0,Y 363.902,Z 398.437,A -85,B 0,C 180,E1 12937.802,E2 12937.802} C_VEL
LIN {X 0,Y 368.896,Z 415.425,A -85,B 0,C 180,E1 12934.752,E2 12934.752} C_VEL
LIN {X 0,Y 347.702,Z 578.804,A -85,B 0,C 180,E1 12930.386,E2 12930.386} C_VEL
LIN {X 0,Y 343.26,Z 640.84,A -85,B 0,C 180,E1 12929.077,E2 12929.077} C_VEL
LIN {X 0,Y 339.632,Z 674.063,A -85,B 0,C 180,E1 12928.177,E2 12928.177} C_VEL
LIN {X 0,Y 334.92,Z 706.612,A -85,B 0,C 180,E1 12927.069,E2 12927.069} C_VEL
LIN {X 0,Y 329.773,Z 736.672,A -85,B 0,C 180,E1 12925.791,E2 12925.791} C_VEL
LIN {X 0,Y 324.267,Z 764.925,A -85,B 0,C 180,E1 12924.266,E2 12924.266} C_VEL
LIN {X 0,Y 318.05,Z 793.74,A -85,B 0,C 180,E1 12922.395,E2 12922.395} C_VEL
LIN {X 0,Y 313.326,Z 813.545,A -85,B 0,C 180,E1 12920.847,E2 12920.847} C_VEL
LIN {X 0,Y 308.022,Z 832.534,A -85,B 0,C 180,E1 12919.002,E2 12919.002} C_VEL
LIN {X 0,Y 302.499,Z 849.927,A -85,B 0,C 180,E1 12916.928,E2 12916.928} C_VEL
LIN {X 0,Y 296.599,Z 866.61,A -85,B 0,C 180,E1 12914.524,E2 12914.524} C_VEL
LIN {X 0,Y 290.406,Z 882.917,A -85,B 0,C 180,E1 12911.645,E2 12911.645} C_VEL
LIN {X 0,Y 284.535,Z 897.684,A -85,B 0,C 180,E1 12908.462,E2 12908.462} C_VEL
LIN {X 0,Y 278.87,Z 911.797,A -85,B 0,C 180,E1 12904.757,E2 12904.757} C_VEL
LIN {X 0,Y 274.014,Z 924.334,A -85,B 0,C 180,E1 12900.721,E2 12900.721} C_VEL
LIN {X 0,Y 270.15,Z 935.188,A -85,B 0,C 180,E1 12896.369,E2 12896.369} C_VEL
LIN {X 0,Y 267.426,Z 944.444,A -85,B 0,C 180,E1 12891.725,E2 12891.725} C_VEL
LIN {X 0,Y 265.952,Z 951.758,A -85,B 0,C 180,E1 12887.053,E2 12887.053} C_VEL
LIN {X 0,Y 265.54,Z 957.219,A -85,B 0,C 180,E1 12882.394,E2 12882.394} C_VEL
LIN {X 0,Y 265.804,Z 960.804,A -85,B 0,C 180,E1 12878.001,E2 12878.001} C_VEL
LIN {X 0,Y 266.299,Z 962.817,A -85,B 0,C 180,E1 12873.875,E2 12873.875} C_VEL
LIN {X 0,Y 266.367,Z 964.649,A -85,B 0,C 180,E1 12870,E2 12870} C_VEL
LIN {X 0,Y 266.018,Z 965.374,A -85,B 0,C 180,E1 12866.552,E2 12866.552} C_VEL
LIN {X 0,Y 265.461,Z 965.112,A -85,B 0,C 180,E1 12862.86,E2 12862.86} C_VEL
LIN {X 0,Y 265.046,Z 963.601,A -85,B 0,C 180,E1 12858.466,E2 12858.466} C_VEL
LIN {X 0,Y 265.547,Z 959.968,A -85,B 0,C 180,E1 12852.92,E2 12852.92} C_VEL
LIN {X 0,Y 267.446,Z 955.13,A -85,B 0,C 180,E1 12847.814,E2 12847.814} C_VEL
LIN {X 0,Y 272.085,Z 947.409,A -85,B 0,C 180,E1 12841.701,E2 12841.701} C_VEL
LIN {X 0,Y 279.501,Z 937.848,A -85,B 0,C 180,E1 12835.83,E2 12835.83} C_VEL
LIN {X 0,Y 289.909,Z 926.294,A -85,B 0,C 180,E1 12830.275,E2 12830.275} C_VEL
LIN {X 0,Y 304.431,Z 911.944,A -85,B 0,C 180,E1 12824.81,E2 12824.81} C_VEL
LIN {X 0,Y 321.084,Z 896.78,A -85,B 0,C 180,E1 12820.274,E2 12820.274} C_VEL
LIN {X 0,Y 335.98,Z 883.69,A -85,B 0,C 180,E1 12817.113,E2 12817.113} C_VEL
LIN {X 0,Y 320.197,Z 893.303,A -85,B 0,C 180,E1 12813.769,E2 12813.769} C_VEL
LIN {X 0,Y 306.371,Z 901.354,A -85,B 0,C 180,E1 12809.956,E2 12809.956} C_VEL
LIN {X 0,Y 295.108,Z 907.303,A -85,B 0,C 180,E1 12805.918,E2 12805.918} C_VEL
LIN {X 0,Y 286.494,Z 911.032,A -85,B 0,C 180,E1 12801.928,E2 12801.928} C_VEL
LIN {X 0,Y 279.523,Z 912.961,A -85,B 0,C 180,E1 12797.701,E2 12797.701} C_VEL
LIN {X 0,Y 274.597,Z 913.028,A -85,B 0,C 180,E1 12793.691,E2 12793.691} C_VEL
LIN {X 0,Y 270.967,Z 911.374,A -85,B 0,C 180,E1 12789.558,E2 12789.558} C_VEL
LIN {X 0,Y 268.494,Z 907.861,A -85,B 0,C 180,E1 12785.342,E2 12785.342} C_VEL
LIN {X 0,Y 267.113,Z 902.722,A -85,B 0,C 180,E1 12781.287,E2 12781.287} C_VEL
LIN {X 0,Y 266.496,Z 895.934,A -85,B 0,C 180,E1 12777.305,E2 12777.305} C_VEL
LIN {X 0,Y 266.5,Z 887.774,A -85,B 0,C 180,E1 12773.537,E2 12773.537} C_VEL
LIN {X 0,Y 267.095,Z 877.385,A -85,B 0,C 180,E1 12769.648,E2 12769.648} C_VEL
LIN {X 0,Y 268.276,Z 865.508,A -85,B 0,C 180,E1 12765.98,E2 12765.98} C_VEL
LIN {X 0,Y 270.015,Z 852.195,A -85,B 0,C 180,E1 12762.545,E2 12762.545} C_VEL
LIN {X 0,Y 272.488,Z 835.962,A -85,B 0,C 180,E1 12759.036,E2 12759.036} C_VEL
LIN {X 0,Y 275.487,Z 817.977,A -85,B 0,C 180,E1 12755.786,E2 12755.786} C_VEL
LIN {X 0,Y 278.801,Z 798.85,A -85,B 0,C 180,E1 12752.904,E2 12752.904} C_VEL
LIN {X 0,Y 282.236,Z 778.557,A -85,B 0,C 180,E1 12750.382,E2 12750.382} C_VEL
LIN {X 0,Y 285.146,Z 761.379,A -85,B 0,C 180,E1 12748.543,E2 12748.543} C_VEL
LIN {X 0,Y 286.729,Z 761.147,A -85,B 0,C 180,E1 12747.99,E2 12747.99} C_VEL
LIN {X 0,Y 289.74,Z 758.909,A -85,B 0,C 180,E1 12747.357,E2 12747.357} C_VEL
LIN {X 0,Y 294.315,Z 754.082,A -85,B 0,C 180,E1 12746.724,E2 12746.724} C_VEL
LIN {X 0,Y 297.283,Z 752.301,A -85,B 0,C 180,E1 12746.059,E2 12746.059} C_VEL
LIN {X 0,Y 301.725,Z 748.238,A -85,B 0,C 180,E1 12745.365,E2 12745.365} C_VEL
LIN {X 0,Y 305.43,Z 743.832,A -85,B 0,C 180,E1 12744.944,E2 12744.944} C_VEL
LIN {X 0,Y 309.582,Z 740.494,A -85,B 0,C 180,E1 12744.225,E2 12744.225} C_VEL
LIN {X 0,Y 314.388,Z 735.324,A -85,B 0,C 180,E1 12743.63,E2 12743.63} C_VEL
LIN {X 0,Y 318.866,Z 729.325,A -85,B 0,C 180,E1 12743.206,E2 12743.206} C_VEL
LIN {X 0,Y 324.23,Z 723.906,A -85,B 0,C 180,E1 12742.478,E2 12742.478} C_VEL
LIN {X 0,Y 329.942,Z 716.128,A -85,B 0,C 180,E1 12741.923,E2 12741.923} C_VEL
LIN {X 0,Y 334.161,Z 709.076,A -85,B 0,C 180,E1 12741.625,E2 12741.625} C_VEL
LIN {X 0,Y 339.511,Z 702.211,A -85,B 0,C 180,E1 12741.004,E2 12741.004} C_VEL
LIN {X 0,Y 340.39,Z 701.1,A -85,B 0,C 180,E1 12740.902,E2 12740.902} C_VEL
LIN {X 0,Y 336.602,Z 721.861,A -85,B 0,C 180,E1 12739.768,E2 12739.768} C_VEL
LIN {X 0,Y 331.63,Z 743.031,A -85,B 0,C 180,E1 12738.302,E2 12738.302} C_VEL
LIN {X 0,Y 326.08,Z 762.53,A -85,B 0,C 180,E1 12736.614,E2 12736.614} C_VEL
LIN {X 0,Y 319.86,Z 781.204,A -85,B 0,C 180,E1 12734.629,E2 12734.629} C_VEL
LIN {X 0,Y 313.009,Z 799.27,A -85,B 0,C 180,E1 12732.279,E2 12732.279} C_VEL
LIN {X 0,Y 305.9,Z 816.106,A -85,B 0,C 180,E1 12729.598,E2 12729.598} C_VEL
LIN {X 0,Y 298.762,Z 831.616,A -85,B 0,C 180,E1 12726.565,E2 12726.565} C_VEL
LIN {X 0,Y 291.947,Z 845.488,A -85,B 0,C 180,E1 12723.229,E2 12723.229} C_VEL
LIN {X 0,Y 285.632,Z 857.785,A -85,B 0,C 180,E1 12719.577,E2 12719.577} C_VEL
LIN {X 0,Y 280.009,Z 868.505,A -85,B 0,C 180,E1 12715.6,E2 12715.6} C_VEL
LIN {X 0,Y 275.246,Z 877.627,A -85,B 0,C 180,E1 12711.301,E2 12711.301} C_VEL
LIN {X 0,Y 271.595,Z 884.884,A -85,B 0,C 180,E1 12706.822,E2 12706.822} C_VEL
LIN {X 0,Y 268.992,Z 890.399,A -85,B 0,C 180,E1 12702.144,E2 12702.144} C_VEL
LIN {X 0,Y 267.473,Z 893.986,A -85,B 0,C 180,E1 12697.518,E2 12697.518} C_VEL
LIN {X 0,Y 266.772,Z 895.828,A -85,B 0,C 180,E1 12693.008,E2 12693.008} C_VEL
LIN {X 0,Y 266.662,Z 896.121,A -85,B 0,C 180,E1 12688.711,E2 12688.711} C_VEL
LIN {X 0,Y 267.113,Z 894.908,A -85,B 0,C 180,E1 12684.199,E2 12684.199} C_VEL
LIN {X 0,Y 268.239,Z 892.115,A -85,B 0,C 180,E1 12679.693,E2 12679.693} C_VEL
LIN {X 0,Y 270.266,Z 887.671,A -85,B 0,C 180,E1 12675.21,E2 12675.21} C_VEL
LIN {X 0,Y 273.328,Z 881.472,A -85,B 0,C 180,E1 12670.778,E2 12670.778} C_VEL
LIN {X 0,Y 277.515,Z 873.376,A -85,B 0,C 180,E1 12666.426,E2 12666.426} C_VEL
LIN {X 0,Y 282.598,Z 863.747,A -85,B 0,C 180,E1 12662.387,E2 12662.387} C_VEL
LIN {X 0,Y 288.734,Z 851.984,A -85,B 0,C 180,E1 12658.472,E2 12658.472} C_VEL
LIN {X 0,Y 295.141,Z 839.32,A -85,B 0,C 180,E1 12655.071,E2 12655.071} C_VEL
LIN {X 0,Y 301.919,Z 825.203,A -85,B 0,C 180,E1 12651.976,E2 12651.976} C_VEL
LIN {X 0,Y 308.9,Z 809.554,A -85,B 0,C 180,E1 12649.167,E2 12649.167} C_VEL
LIN {X 0,Y 315.928,Z 792.228,A -85,B 0,C 180,E1 12646.624,E2 12646.624} C_VEL
LIN {X 0,Y 322.368,Z 774.489,A -85,B 0,C 180,E1 12644.489,E2 12644.489} C_VEL
LIN {X 0,Y 328.282,Z 755.819,A -85,B 0,C 180,E1 12642.645,E2 12642.645} C_VEL
LIN {X 0,Y 333.552,Z 736.201,A -85,B 0,C 180,E1 12641.069,E2 12641.069} C_VEL
LIN {X 0,Y 338.068,Z 715.486,A -85,B 0,C 180,E1 12639.737,E2 12639.737} C_VEL
LIN {X 0,Y 341.601,Z 694.386,A -85,B 0,C 180,E1 12638.675,E2 12638.675} C_VEL
LIN {X 0,Y 345.016,Z 671.14,A -85,B 0,C 180,E1 12637.707,E2 12637.707} C_VEL
LIN {X 0,Y 345.559,Z 663.804,A -85,B 0,C 180,E1 12637.291,E2 12637.291} C_VEL
LIN {X 0,Y 344.886,Z 645.737,A -85,B 0,C 180,E1 12635.826,E2 12635.826} C_VEL
LIN {X 0,Y 345.461,Z 638.348,A -85,B 0,C 180,E1 12635.453,E2 12635.453} C_VEL
LIN {X 0,Y 352.686,Z 589.505,A -85,B 0,C 180,E1 12634.08,E2 12634.08} C_VEL
LIN {X 0,Y 358.626,Z 541.142,A -85,B 0,C 180,E1 12632.942,E2 12632.942} C_VEL
LIN {X 0,Y 363.158,Z 492.249,A -85,B 0,C 180,E1 12631.98,E2 12631.98} C_VEL
LIN {X 0,Y 366.865,Z 447.449,A -85,B 0,C 180,E1 12631.172,E2 12631.172} C_VEL
LIN {X 0,Y 372.743,Z 422.289,A -85,B 0,C 180,E1 12630.375,E2 12630.375} C_VEL
LIN {X 0,Y 368.415,Z 408.009,A -85,B 0,C 180,E1 12627.389,E2 12627.389} C_VEL
LIN {X 0,Y 364.236,Z 395.66,A -85,B 0,C 180,E1 12624.36,E2 12624.36} C_VEL
LIN {X 0,Y 360.156,Z 384.746,A -85,B 0,C 180,E1 12621.157,E2 12621.157} C_VEL
LIN {X 0,Y 356.22,Z 374.962,A -85,B 0,C 180,E1 12617.689,E2 12617.689} C_VEL
LIN {X 0,Y 352.759,Z 366.756,A -85,B 0,C 180,E1 12614.025,E2 12614.025} C_VEL
LIN {X 0,Y 350.734,Z 362.044,A -85,B 0,C 180,E1 12611.278,E2 12611.278} C_VEL
LIN {X 0,Y 349.13,Z 358.063,A -85,B 0,C 180,E1 12608.565,E2 12608.565} C_VEL
LIN {X 0,Y 347.607,Z 354.308,A -85,B 0,C 180,E1 12605.033,E2 12605.033} C_VEL
LIN {X 0,Y 347.482,Z 353.459,A -85,B 0,C 180,E1 12604.125,E2 12604.125} C_VEL
LIN {X 0,Y 347.085,Z 352.111,A -85,B 0,C 180,E1 12598.184,E2 12598.184} C_VEL
LIN {X 0,Y 349.109,Z 353.469,A -85,B 0,C 180,E1 12593.091,E2 12593.091} C_VEL
LIN {X 0,Y 349.322,Z 353.983,A -85,B 0,C 180,E1 12592.641,E2 12592.641} C_VEL
LIN {X 0,Y 350.507,Z 364.551,A -85,B 0,C 180,E1 12588.981,E2 12588.981} C_VEL
LIN {X 0,Y 352.914,Z 376.48,A -85,B 0,C 180,E1 12585.353,E2 12585.353} C_VEL
LIN {X 0,Y 358.177,Z 395.672,A -85,B 0,C 180,E1 12580.428,E2 12580.428} C_VEL
LIN {X 0,Y 361.075,Z 404.965,A -85,B 0,C 180,E1 12578.389,E2 12578.389} C_VEL
LIN {X 0,Y 364.976,Z 419.19,A -85,B 0,C 180,E1 12575.794,E2 12575.794} C_VEL
LIN {X 0,Y 343.906,Z 575.914,A -85,B 0,C 180,E1 12571.605,E2 12571.605} C_VEL
LIN {X 0,Y 339.36,Z 637.568,A -85,B 0,C 180,E1 12570.3,E2 12570.3} C_VEL
LIN {X 0,Y 335.582,Z 671.204,A -85,B 0,C 180,E1 12569.4,E2 12569.4} C_VEL
LIN {X 0,Y 330.753,Z 703.669,A -85,B 0,C 180,E1 12568.31,E2 12568.31} C_VEL
LIN {X 0,Y 325.385,Z 734.286,A -85,B 0,C 180,E1 12567.025,E2 12567.025} C_VEL
LIN {X 0,Y 319.944,Z 761.293,A -85,B 0,C 180,E1 12565.594,E2 12565.594} C_VEL
LIN {X 0,Y 313.887,Z 788.844,A -85,B 0,C 180,E1 12563.855,E2 12563.855} C_VEL
LIN {X 0,Y 308.688,Z 810.28,A -85,B 0,C 180,E1 12562.219,E2 12562.219} C_VEL
LIN {X 0,Y 303.137,Z 829.589,A -85,B 0,C 180,E1 12560.371,E2 12560.371} C_VEL
LIN {X 0,Y 297.3,Z 847.226,A -85,B 0,C 180,E1 12558.3,E2 12558.3} C_VEL
LIN {X 0,Y 290.87,Z 864.744,A -85,B 0,C 180,E1 12555.786,E2 12555.786} C_VEL
LIN {X 0,Y 284.444,Z 880.988,A -85,B 0,C 180,E1 12552.911,E2 12552.911} C_VEL
LIN {X 0,Y 278.335,Z 895.629,A -85,B 0,C 180,E1 12549.75,E2 12549.75} C_VEL
LIN {X 0,Y 272.276,Z 909.882,A -85,B 0,C 180,E1 12545.985,E2 12545.985} C_VEL
LIN {X 0,Y 267.294,Z 921.921,A -85,B 0,C 180,E1 12542.086,E2 12542.086} C_VEL
LIN {X 0,Y 263.198,Z 932.582,A -85,B 0,C 180,E1 12537.858,E2 12537.858} C_VEL
LIN {X 0,Y 260.13,Z 941.834,A -85,B 0,C 180,E1 12533.267,E2 12533.267} C_VEL
LIN {X 0,Y 258.224,Z 949.726,A -85,B 0,C 180,E1 12528.279,E2 12528.279} C_VEL
LIN {X 0,Y 257.569,Z 955.485,A -85,B 0,C 180,E1 12523.469,E2 12523.469} C_VEL
LIN {X 0,Y 257.778,Z 959.51,A -85,B 0,C 180,E1 12518.701,E2 12518.701} C_VEL
LIN {X 0,Y 258.287,Z 961.671,A -85,B 0,C 180,E1 12514.44,E2 12514.44} C_VEL
LIN {X 0,Y 258.519,Z 962.811,A -85,B 0,C 180,E1 12511.108,E2 12511.108} C_VEL
LIN {X 0,Y 258.193,Z 964.018,A -85,B 0,C 180,E1 12507.114,E2 12507.114} C_VEL
LIN {X 0,Y 257.543,Z 963.94,A -85,B 0,C 180,E1 12502.863,E2 12502.863} C_VEL
LIN {X 0,Y 257.104,Z 962.669,A -85,B 0,C 180,E1 12498.534,E2 12498.534} C_VEL
LIN {X 0,Y 257.44,Z 959.909,A -85,B 0,C 180,E1 12493.529,E2 12493.529} C_VEL
LIN {X 0,Y 259.646,Z 954.661,A -85,B 0,C 180,E1 12487.35,E2 12487.35} C_VEL
LIN {X 0,Y 264.211,Z 947.807,A -85,B 0,C 180,E1 12481.401,E2 12481.401} C_VEL
LIN {X 0,Y 272.006,Z 938.514,A -85,B 0,C 180,E1 12475.265,E2 12475.265} C_VEL
LIN {X 0,Y 283.522,Z 926.959,A -85,B 0,C 180,E1 12469.274,E2 12469.274} C_VEL
LIN {X 0,Y 298.295,Z 913.641,A -85,B 0,C 180,E1 12463.889,E2 12463.889} C_VEL
LIN {X 0,Y 315.481,Z 899.188,A -85,B 0,C 180,E1 12459.337,E2 12459.337} C_VEL
LIN {X 0,Y 326.168,Z 890.562,A -85,B 0,C 180,E1 12457.052,E2 12457.052} C_VEL
LIN {X 0,Y 310.014,Z 899.337,A -85,B 0,C 180,E1 12453.472,E2 12453.472} C_VEL
LIN {X 0,Y 296.356,Z 906.225,A -85,B 0,C 180,E1 12449.512,E2 12449.512} C_VEL
LIN {X 0,Y 285.264,Z 911.069,A -85,B 0,C 180,E1 12445.317,E2 12445.317} C_VEL
LIN {X 0,Y 276.501,Z 913.864,A -85,B 0,C 180,E1 12440.978,E2 12440.978} C_VEL
LIN {X 0,Y 269.849,Z 914.678,A -85,B 0,C 180,E1 12436.578,E2 12436.578} C_VEL
LIN {X 0,Y 265.25,Z 913.719,A -85,B 0,C 180,E1 12432.408,E2 12432.408} C_VEL
LIN {X 0,Y 261.959,Z 911.019,A -85,B 0,C 180,E1 12428.119,E2 12428.119} C_VEL
LIN {X 0,Y 259.841,Z 906.46,A -85,B 0,C 180,E1 12423.751,E2 12423.751} C_VEL
LIN {X 0,Y 258.767,Z 900.288,A -85,B 0,C 180,E1 12419.557,E2 12419.557} C_VEL
LIN {X 0,Y 258.435,Z 892.664,A -85,B 0,C 180,E1 12415.562,E2 12415.562} C_VEL
LIN {X 0,Y 258.727,Z 883.15,A -85,B 0,C 180,E1 12411.555,E2 12411.555} C_VEL
LIN {X 0,Y 259.6,Z 872.174,A -85,B 0,C 180,E1 12407.77,E2 12407.77} C_VEL
LIN {X 0,Y 261.198,Z 858.773,A -85,B 0,C 180,E1 12403.916,E2 12403.916} C_VEL
LIN {X 0,Y 263.291,Z 844.477,A -85,B 0,C 180,E1 12400.476,E2 12400.476} C_VEL
LIN {X 0,Y 266.029,Z 827.779,A -85,B 0,C 180,E1 12397.107,E2 12397.107} C_VEL
LIN {X 0,Y 269.345,Z 808.814,A -85,B 0,C 180,E1 12393.902,E2 12393.902} C_VEL
LIN {X 0,Y 272.919,Z 788.641,A -85,B 0,C 180,E1 12391.079,E2 12391.079} C_VEL
LIN {X 0,Y 275.484,Z 774.071,A -85,B 0,C 180,E1 12389.309,E2 12389.309} C_VEL
LIN {X 0,Y 277.117,Z 773.825,A -85,B 0,C 180,E1 12388.696,E2 12388.696} C_VEL
LIN {X 0,Y 279.822,Z 772.019,A -85,B 0,C 180,E1 12388.072,E2 12388.072} C_VEL
LIN {X 0,Y 283.993,Z 768.125,A -85,B 0,C 180,E1 12387.405,E2 12387.405} C_VEL
LIN {X 0,Y 287.484,Z 766.13,A -85,B 0,C 180,E1 12386.589,E2 12386.589} C_VEL
LIN {X 0,Y 292.129,Z 762.099,A -85,B 0,C 180,E1 12385.852,E2 12385.852} C_VEL
LIN {X 0,Y 293.991,Z 760.179,A -85,B 0,C 180,E1 12385.627,E2 12385.627} C_VEL
LIN {X 0,Y 298.345,Z 757.201,A -85,B 0,C 180,E1 12384.798,E2 12384.798} C_VEL
LIN {X 0,Y 303.846,Z 751.934,A -85,B 0,C 180,E1 12384.051,E2 12384.051} C_VEL
LIN {X 0,Y 306.307,Z 749.242,A -85,B 0,C 180,E1 12383.783,E2 12383.783} C_VEL
LIN {X 0,Y 311.901,Z 744.537,A -85,B 0,C 180,E1 12382.963,E2 12382.963} C_VEL
LIN {X 0,Y 317.585,Z 738.191,A -85,B 0,C 180,E1 12382.353,E2 12382.353} C_VEL
LIN {X 0,Y 320.622,Z 734.323,A -85,B 0,C 180,E1 12382.094,E2 12382.094} C_VEL
LIN {X 0,Y 326.669,Z 728.199,A -85,B 0,C 180,E1 12381.36,E2 12381.36} C_VEL
LIN {X 0,Y 331.79,Z 721.533,A -85,B 0,C 180,E1 12380.9,E2 12380.9} C_VEL
LIN {X 0,Y 327.148,Z 741.267,A -85,B 0,C 180,E1 12379.556,E2 12379.556} C_VEL
LIN {X 0,Y 321.749,Z 760.218,A -85,B 0,C 180,E1 12377.965,E2 12377.965} C_VEL
LIN {X 0,Y 315.427,Z 779.078,A -85,B 0,C 180,E1 12376.02,E2 12376.02} C_VEL
LIN {X 0,Y 308.575,Z 796.943,A -85,B 0,C 180,E1 12373.761,E2 12373.761} C_VEL
LIN {X 0,Y 301.421,Z 813.63,A -85,B 0,C 180,E1 12371.184,E2 12371.184} C_VEL
LIN {X 0,Y 294.083,Z 829.245,A -85,B 0,C 180,E1 12368.229,E2 12368.229} C_VEL
LIN {X 0,Y 287.194,Z 842.907,A -85,B 0,C 180,E1 12365.062,E2 12365.062} C_VEL
LIN {X 0,Y 280.689,Z 855.168,A -85,B 0,C 180,E1 12361.578,E2 12361.578} C_VEL
LIN {X 0,Y 274.762,Z 866.016,A -85,B 0,C 180,E1 12357.763,E2 12357.763} C_VEL
LIN {X 0,Y 269.581,Z 875.414,A -85,B 0,C 180,E1 12353.614,E2 12353.614} C_VEL
LIN {X 0,Y 265.321,Z 883.278,A -85,B 0,C 180,E1 12349.14,E2 12349.14} C_VEL
LIN {X 0,Y 262.232,Z 889.286,A -85,B 0,C 180,E1 12344.576,E2 12344.576} C_VEL
LIN {X 0,Y 260.213,Z 893.564,A -85,B 0,C 180,E1 12339.958,E2 12339.958} C_VEL
LIN {X 0,Y 259.111,Z 896.158,A -85,B 0,C 180,E1 12335.314,E2 12335.314} C_VEL
LIN {X 0,Y 258.716,Z 897.151,A -85,B 0,C 180,E1 12330.886,E2 12330.886} C_VEL
LIN {X 0,Y 258.893,Z 896.681,A -85,B 0,C 180,E1 12326.236,E2 12326.236} C_VEL
LIN {X 0,Y 259.735,Z 894.645,A -85,B 0,C 180,E1 12321.588,E2 12321.588} C_VEL
LIN {X 0,Y 261.405,Z 891.002,A -85,B 0,C 180,E1 12316.957,E2 12316.957} C_VEL
LIN {X 0,Y 264.12,Z 885.658,A -85,B 0,C 180,E1 12312.371,E2 12312.371} C_VEL
LIN {X 0,Y 267.957,Z 878.492,A -85,B 0,C 180,E1 12307.859,E2 12307.859} C_VEL
LIN {X 0,Y 272.742,Z 869.847,A -85,B 0,C 180,E1 12303.667,E2 12303.667} C_VEL
LIN {X 0,Y 278.618,Z 859.197,A -85,B 0,C 180,E1 12299.601,E2 12299.601} C_VEL
LIN {X 0,Y 285.198,Z 846.976,A -85,B 0,C 180,E1 12295.878,E2 12295.878} C_VEL
LIN {X 0,Y 292.279,Z 833.18,A -85,B 0,C 180,E1 12292.487,E2 12292.487} C_VEL
LIN {X 0,Y 299.457,Z 818.252,A -85,B 0,C 180,E1 12289.501,E2 12289.501} C_VEL
LIN {X 0,Y 306.505,Z 802.316,A -85,B 0,C 180,E1 12286.887,E2 12286.887} C_VEL
LIN {X 0,Y 313.469,Z 784.852,A -85,B 0,C 180,E1 12284.541,E2 12284.541} C_VEL
LIN {X 0,Y 319.752,Z 767.032,A -85,B 0,C 180,E1 12282.572,E2 12282.572} C_VEL
LIN {X 0,Y 325.624,Z 747.606,A -85,B 0,C 180,E1 12280.82,E2 12280.82} C_VEL
LIN {X 0,Y 330.583,Z 728.05,A -85,B 0,C 180,E1 12279.395,E2 12279.395} C_VEL
LIN {X 0,Y 334.804,Z 706.92,A -85,B 0,C 180,E1 12278.17,E2 12278.17} C_VEL
LIN {X 0,Y 340.845,Z 668.017,A -85,B 0,C 180,E1 12276.488,E2 12276.488} C_VEL
LIN {X 0,Y 345.461,Z 638.348,A -85,B 0,C 180,E1 12275.453,E2 12275.453} C_VEL
LIN {X 0,Y 346.093,Z 630.92,A -85,B 0,C 180,E1 12275.092,E2 12275.092} C_VEL
LIN {X 0,Y 345.73,Z 611.532,A -85,B 0,C 180,E1 12273.656,E2 12273.656} C_VEL
LIN {X 0,Y 346.295,Z 605.133,A -85,B 0,C 180,E1 12273.369,E2 12273.369} C_VEL
LIN {X 0,Y 352.764,Z 556.34,A -85,B 0,C 180,E1 12272.17,E2 12272.17} C_VEL
LIN {X 0,Y 357.731,Z 508.112,A -85,B 0,C 180,E1 12271.178,E2 12271.178} C_VEL
LIN {X 0,Y 362.648,Z 450.247,A -85,B 0,C 180,E1 12270.129,E2 12270.129} C_VEL
LIN {X 0,Y 368.302,Z 426.072,A -85,B 0,C 180,E1 12269.37,E2 12269.37} C_VEL
LIN {X 0,Y 364.176,Z 412.156,A -85,B 0,C 180,E1 12266.366,E2 12266.366} C_VEL
LIN {X 0,Y 360.093,Z 399.779,A -85,B 0,C 180,E1 12263.179,E2 12263.179} C_VEL
LIN {X 0,Y 356.102,Z 388.919,A -85,B 0,C 180,E1 12259.819,E2 12259.819} C_VEL
LIN {X 0,Y 352.793,Z 380.573,A -85,B 0,C 180,E1 12256.634,E2 12256.634} C_VEL
LIN {X 0,Y 350.053,Z 373.712,A -85,B 0,C 180,E1 12253.462,E2 12253.462} C_VEL
LIN {X 0,Y 348.405,Z 369.611,A -85,B 0,C 180,E1 12251.086,E2 12251.086} C_VEL
LIN {X 0,Y 346.952,Z 365.624,A -85,B 0,C 180,E1 12248.285,E2 12248.285} C_VEL
LIN {X 0,Y 345.586,Z 361.831,A -85,B 0,C 180,E1 12244.73,E2 12244.73} C_VEL
LIN {X 0,Y 345.451,Z 361.14,A -85,B 0,C 180,E1 12243.817,E2 12243.817} C_VEL
LIN {X 0,Y 345.294,Z 359.908,A -85,B 0,C 180,E1 12238.175,E2 12238.175} C_VEL
LIN {X 0,Y 347.292,Z 361.192,A -85,B 0,C 180,E1 12233.359,E2 12233.359} C_VEL
LIN {X 0,Y 347.467,Z 361.736,A -85,B 0,C 180,E1 12232.934,E2 12232.934} C_VEL
LIN {X 0,Y 348.421,Z 371.605,A -85,B 0,C 180,E1 12229.5,E2 12229.5} C_VEL
LIN {X 0,Y 350.524,Z 383.357,A -85,B 0,C 180,E1 12225.899,E2 12225.899} C_VEL
LIN {X 0,Y 355.377,Z 401.98,A -85,B 0,C 180,E1 12221.079,E2 12221.079} C_VEL
LIN {X 0,Y 358.077,Z 411.08,A -85,B 0,C 180,E1 12219.058,E2 12219.058} C_VEL
LIN {X 0,Y 361.157,Z 423.112,A -85,B 0,C 180,E1 12216.855,E2 12216.855} C_VEL
LIN {X 0,Y 340.28,Z 572.859,A -85,B 0,C 180,E1 12212.853,E2 12212.853} C_VEL
LIN {X 0,Y 335.724,Z 633.339,A -85,B 0,C 180,E1 12211.575,E2 12211.575} C_VEL
LIN {X 0,Y 331.756,Z 667.831,A -85,B 0,C 180,E1 12210.666,E2 12210.666} C_VEL
LIN {X 0,Y 326.687,Z 701.265,A -85,B 0,C 180,E1 12209.56,E2 12209.56} C_VEL
LIN {X 0,Y 321.248,Z 731.396,A -85,B 0,C 180,E1 12208.32,E2 12208.32} C_VEL
LIN {X 0,Y 315.648,Z 758.328,A -85,B 0,C 180,E1 12206.915,E2 12206.915} C_VEL
LIN {X 0,Y 309.661,Z 785.042,A -85,B 0,C 180,E1 12205.263,E2 12205.263} C_VEL
LIN {X 0,Y 304.091,Z 807.531,A -85,B 0,C 180,E1 12203.576,E2 12203.576} C_VEL
LIN {X 0,Y 298.703,Z 825.778,A -85,B 0,C 180,E1 12201.873,E2 12201.873} C_VEL
LIN {X 0,Y 292.289,Z 844.528,A -85,B 0,C 180,E1 12199.717,E2 12199.717} C_VEL
LIN {X 0,Y 285.621,Z 862.049,A -85,B 0,C 180,E1 12197.223,E2 12197.223} C_VEL
LIN {X 0,Y 278.897,Z 878.424,A -85,B 0,C 180,E1 12194.355,E2 12194.355} C_VEL
LIN {X 0,Y 272.274,Z 893.536,A -85,B 0,C 180,E1 12191.098,E2 12191.098} C_VEL
LIN {X 0,Y 266.16,Z 907.221,A -85,B 0,C 180,E1 12187.487,E2 12187.487} C_VEL
LIN {X 0,Y 260.454,Z 920.133,A -85,B 0,C 180,E1 12183.297,E2 12183.297} C_VEL
LIN {X 0,Y 256.003,Z 930.92,A -85,B 0,C 180,E1 12178.967,E2 12178.967} C_VEL
LIN {X 0,Y 252.644,Z 940.22,A -85,B 0,C 180,E1 12174.305,E2 12174.305} C_VEL
LIN {X 0,Y 250.518,Z 947.999,A -85,B 0,C 180,E1 12169.346,E2 12169.346} C_VEL
LIN {X 0,Y 249.63,Z 954.104,A -85,B 0,C 180,E1 12164.226,E2 12164.226} C_VEL
LIN {X 0,Y 249.741,Z 958.149,A -85,B 0,C 180,E1 12159.448,E2 12159.448} C_VEL
LIN {X 0,Y 250.282,Z 960.475,A -85,B 0,C 180,E1 12155.042,E2 12155.042} C_VEL
LIN {X 0,Y 250.644,Z 961.382,A -85,B 0,C 180,E1 12151.143,E2 12151.143} C_VEL
LIN {X 0,Y 250.335,Z 962.567,A -85,B 0,C 180,E1 12147.253,E2 12147.253} C_VEL
LIN {X 0,Y 249.626,Z 962.76,A -85,B 0,C 180,E1 12142.867,E2 12142.867} C_VEL
LIN {X 0,Y 249.152,Z 961.367,A -85,B 0,C 180,E1 12137.719,E2 12137.719} C_VEL
LIN {X 0,Y 249.664,Z 958.616,A -85,B 0,C 180,E1 12132.52,E2 12132.52} C_VEL
LIN {X 0,Y 252.286,Z 953.52,A -85,B 0,C 180,E1 12126.155,E2 12126.155} C_VEL
LIN {X 0,Y 257.451,Z 946.724,A -85,B 0,C 180,E1 12120.008,E2 12120.008} C_VEL
LIN {X 0,Y 266.746,Z 937.029,A -85,B 0,C 180,E1 12113.338,E2 12113.338} C_VEL
LIN {X 0,Y 279.704,Z 925.495,A -85,B 0,C 180,E1 12107.217,E2 12107.217} C_VEL
LIN {X 0,Y 295.674,Z 912.532,A -85,B 0,C 180,E1 12101.928,E2 12101.928} C_VEL
LIN {X 0,Y 314.698,Z 898.105,A -85,B 0,C 180,E1 12097.363,E2 12097.363} C_VEL
LIN {X 0,Y 316.287,Z 896.898,A -85,B 0,C 180,E1 12096.99,E2 12096.99} C_VEL
LIN {X 0,Y 300.022,Z 904.665,A -85,B 0,C 180,E1 12093.226,E2 12093.226} C_VEL
LIN {X 0,Y 286.291,Z 910.541,A -85,B 0,C 180,E1 12089.043,E2 12089.043} C_VEL
LIN {X 0,Y 275.39,Z 914.302,A -85,B 0,C 180,E1 12084.68,E2 12084.68} C_VEL
LIN {X 0,Y 266.856,Z 916.048,A -85,B 0,C 180,E1 12080.165,E2 12080.165} C_VEL
LIN {X 0,Y 260.728,Z 915.908,A -85,B 0,C 180,E1 12075.8,E2 12075.8} C_VEL
LIN {X 0,Y 256.348,Z 914.113,A -85,B 0,C 180,E1 12071.474,E2 12071.474} C_VEL
LIN {X 0,Y 253.172,Z 910.306,A -85,B 0,C 180,E1 12066.805,E2 12066.805} C_VEL
LIN {X 0,Y 251.366,Z 904.758,A -85,B 0,C 180,E1 12062.28,E2 12062.28} C_VEL
LIN {X 0,Y 250.557,Z 897.616,A -85,B 0,C 180,E1 12057.942,E2 12057.942} C_VEL
LIN {X 0,Y 250.486,Z 889.011,A -85,B 0,C 180,E1 12053.813,E2 12053.813} C_VEL
LIN {X 0,Y 251.021,Z 879.044,A -85,B 0,C 180,E1 12049.906,E2 12049.906} C_VEL
LIN {X 0,Y 252.205,Z 867.049,A -85,B 0,C 180,E1 12046.005,E2 12046.005} C_VEL
LIN {X 0,Y 254.132,Z 852.773,A -85,B 0,C 180,E1 12042.128,E2 12042.128} C_VEL
LIN {X 0,Y 256.667,Z 836.908,A -85,B 0,C 180,E1 12038.519,E2 12038.519} C_VEL
LIN {X 0,Y 259.61,Z 820.001,A -85,B 0,C 180,E1 12035.298,E2 12035.298} C_VEL
LIN {X 0,Y 263.068,Z 800.909,A -85,B 0,C 180,E1 12032.25,E2 12032.25} C_VEL
LIN {X 0,Y 265.919,Z 785.589,A -85,B 0,C 180,E1 12030.118,E2 12030.118} C_VEL
LIN {X 0,Y 267.556,Z 785.32,A -85,B 0,C 180,E1 12029.453,E2 12029.453} C_VEL
LIN {X 0,Y 270.953,Z 783.098,A -85,B 0,C 180,E1 12028.645,E2 12028.645} C_VEL
LIN {X 0,Y 273.496,Z 780.839,A -85,B 0,C 180,E1 12028.233,E2 12028.233} C_VEL
LIN {X 0,Y 277.266,Z 778.882,A -85,B 0,C 180,E1 12027.252,E2 12027.252} C_VEL
LIN {X 0,Y 282.111,Z 774.981,A -85,B 0,C 180,E1 12026.433,E2 12026.433} C_VEL
LIN {X 0,Y 283.627,Z 773.906,A -85,B 0,C 180,E1 12026.151,E2 12026.151} C_VEL
LIN {X 0,Y 288,Z 771.06,A -85,B 0,C 180,E1 12025.293,E2 12025.293} C_VEL
LIN {X 0,Y 293.595,Z 766.149,A -85,B 0,C 180,E1 12024.514,E2 12024.514} C_VEL
LIN {X 0,Y 299.852,Z 761.546,A -85,B 0,C 180,E1 12023.48,E2 12023.48} C_VEL
LIN {X 0,Y 305.844,Z 755.879,A -85,B 0,C 180,E1 12022.784,E2 12022.784} C_VEL
LIN {X 0,Y 307.636,Z 754.215,A -85,B 0,C 180,E1 12022.57,E2 12022.57} C_VEL
LIN {X 0,Y 313.568,Z 749.089,A -85,B 0,C 180,E1 12021.784,E2 12021.784} C_VEL
LIN {X 0,Y 319.861,Z 742.293,A -85,B 0,C 180,E1 12021.188,E2 12021.188} C_VEL
LIN {X 0,Y 322.837,Z 738.833,A -85,B 0,C 180,E1 12020.929,E2 12020.929} C_VEL
LIN {X 0,Y 323.024,Z 738.715,A -85,B 0,C 180,E1 12020.899,E2 12020.899} C_VEL
LIN {X 0,Y 317.433,Z 758.321,A -85,B 0,C 180,E1 12019.305,E2 12019.305} C_VEL
LIN {X 0,Y 311.041,Z 777.243,A -85,B 0,C 180,E1 12017.405,E2 12017.405} C_VEL
LIN {X 0,Y 303.938,Z 795.536,A -85,B 0,C 180,E1 12015.15,E2 12015.15} C_VEL
LIN {X 0,Y 296.452,Z 812.676,A -85,B 0,C 180,E1 12012.552,E2 12012.552} C_VEL
LIN {X 0,Y 288.766,Z 828.6,A -85,B 0,C 180,E1 12009.578,E2 12009.578} C_VEL
LIN {X 0,Y 281.516,Z 842.523,A -85,B 0,C 180,E1 12006.381,E2 12006.381} C_VEL
LIN {X 0,Y 274.282,Z 855.624,A -85,B 0,C 180,E1 12002.652,E2 12002.652} C_VEL
LIN {X 0,Y 267.984,Z 866.636,A -85,B 0,C 180,E1 11998.738,E2 11998.738} C_VEL
LIN {X 0,Y 262.335,Z 876.359,A -85,B 0,C 180,E1 11994.363,E2 11994.363} C_VEL
LIN {X 0,Y 257.98,Z 883.994,A -85,B 0,C 180,E1 11989.943,E2 11989.943} C_VEL
LIN {X 0,Y 254.652,Z 890.073,A -85,B 0,C 180,E1 11985.253,E2 11985.253} C_VEL
LIN {X 0,Y 252.375,Z 894.573,A -85,B 0,C 180,E1 11980.27,E2 11980.27} C_VEL
LIN {X 0,Y 251.201,Z 897.161,A -85,B 0,C 180,E1 11975.482,E2 11975.482} C_VEL
LIN {X 0,Y 250.779,Z 898.152,A -85,B 0,C 180,E1 11970.914,E2 11970.914} C_VEL
LIN {X 0,Y 250.968,Z 897.684,A -85,B 0,C 180,E1 11966.117,E2 11966.117} C_VEL
LIN {X 0,Y 251.874,Z 895.635,A -85,B 0,C 180,E1 11961.298,E2 11961.298} C_VEL
LIN {X 0,Y 253.644,Z 892.014,A -85,B 0,C 180,E1 11956.551,E2 11956.551} C_VEL
LIN {X 0,Y 256.519,Z 886.679,A -85,B 0,C 180,E1 11951.83,E2 11951.83} C_VEL
LIN {X 0,Y 260.574,Z 879.522,A -85,B 0,C 180,E1 11947.197,E2 11947.197} C_VEL
LIN {X 0,Y 265.604,Z 870.883,A -85,B 0,C 180,E1 11942.902,E2 11942.902} C_VEL
LIN {X 0,Y 271.76,Z 860.242,A -85,B 0,C 180,E1 11938.749,E2 11938.749} C_VEL
LIN {X 0,Y 278.629,Z 848.026,A -85,B 0,C 180,E1 11934.958,E2 11934.958} C_VEL
LIN {X 0,Y 285.817,Z 834.602,A -85,B 0,C 180,E1 11931.595,E2 11931.595} C_VEL
LIN {X 0,Y 293.217,Z 819.817,A -85,B 0,C 180,E1 11928.582,E2 11928.582} C_VEL
LIN {X 0,Y 300.501,Z 803.968,A -85,B 0,C 180,E1 11925.939,E2 11925.939} C_VEL
LIN {X 0,Y 307.713,Z 786.538,A -85,B 0,C 180,E1 11923.563,E2 11923.563} C_VEL
LIN {X 0,Y 314.433,Z 768.065,A -85,B 0,C 180,E1 11921.506,E2 11921.506} C_VEL
LIN {X 0,Y 320.382,Z 749.009,A -85,B 0,C 180,E1 11919.777,E2 11919.777} C_VEL
LIN {X 0,Y 325.424,Z 729.786,A -85,B 0,C 180,E1 11918.365,E2 11918.365} C_VEL
LIN {X 0,Y 329.778,Z 708.764,A -85,B 0,C 180,E1 11917.134,E2 11917.134} C_VEL
LIN {X 0,Y 336.016,Z 670.139,A -85,B 0,C 180,E1 11915.443,E2 11915.443} C_VEL
LIN {X 0,Y 342.419,Z 630.14,A -85,B 0,C 180,E1 11914.076,E2 11914.076} C_VEL
LIN {X 0,Y 346.295,Z 605.133,A -85,B 0,C 180,E1 11913.369,E2 11913.369} C_VEL
LIN {X 0,Y 346.882,Z 597.672,A -85,B 0,C 180,E1 11913.024,E2 11913.024} C_VEL
LIN {X 0,Y 346.361,Z 578.132,A -85,B 0,C 180,E1 11911.648,E2 11911.648} C_VEL
LIN {X 0,Y 346.837,Z 571.682,A -85,B 0,C 180,E1 11911.387,E2 11911.387} C_VEL
LIN {X 0,Y 352.341,Z 523.727,A -85,B 0,C 180,E1 11910.353,E2 11910.353} C_VEL
LIN {X 0,Y 358.549,Z 453.065,A -85,B 0,C 180,E1 11909.063,E2 11909.063} C_VEL
LIN {X 0,Y 364.031,Z 430.052,A -85,B 0,C 180,E1 11908.371,E2 11908.371} C_VEL
LIN {X 0,Y 360.047,Z 416.391,A -85,B 0,C 180,E1 11905.32,E2 11905.32} C_VEL
LIN {X 0,Y 356.323,Z 404.78,A -85,B 0,C 180,E1 11902.204,E2 11902.204} C_VEL
LIN {X 0,Y 352.921,Z 395.214,A -85,B 0,C 180,E1 11899.144,E2 11899.144} C_VEL
LIN {X 0,Y 349.976,Z 387.363,A -85,B 0,C 180,E1 11896.089,E2 11896.089} C_VEL
LIN {X 0,Y 347.406,Z 380.655,A -85,B 0,C 180,E1 11892.889,E2 11892.889} C_VEL
LIN {X 0,Y 345.934,Z 376.873,A -85,B 0,C 180,E1 11890.66,E2 11890.66} C_VEL
LIN {X 0,Y 344.819,Z 373.303,A -85,B 0,C 180,E1 11888.169,E2 11888.169} C_VEL
LIN {X 0,Y 343.577,Z 369.463,A -85,B 0,C 180,E1 11884.507,E2 11884.507} C_VEL
LIN {X 0,Y 343.43,Z 368.82,A -85,B 0,C 180,E1 11883.505,E2 11883.505} C_VEL
LIN {X 0,Y 343.479,Z 367.699,A -85,B 0,C 180,E1 11878.332,E2 11878.332} C_VEL
LIN {X 0,Y 345.279,Z 368.86,A -85,B 0,C 180,E1 11873.682,E2 11873.682} C_VEL
LIN {X 0,Y 345.488,Z 369.332,A -85,B 0,C 180,E1 11873.269,E2 11873.269} C_VEL
LIN {X 0,Y 346.364,Z 378.658,A -85,B 0,C 180,E1 11870.026,E2 11870.026} C_VEL
LIN {X 0,Y 348.175,Z 390.05,A -85,B 0,C 180,E1 11866.506,E2 11866.506} C_VEL
LIN {X 0,Y 352.845,Z 408.971,A -85,B 0,C 180,E1 11861.581,E2 11861.581} C_VEL
LIN {X 0,Y 355.205,Z 417.496,A -85,B 0,C 180,E1 11859.678,E2 11859.678} C_VEL
LIN {X 0,Y 357.47,Z 426.949,A -85,B 0,C 180,E1 11857.939,E2 11857.939} C_VEL
LIN {X 0,Y 336.817,Z 569.861,A -85,B 0,C 180,E1 11854.126,E2 11854.126} C_VEL
LIN {X 0,Y 332.163,Z 629.931,A -85,B 0,C 180,E1 11852.855,E2 11852.855} C_VEL
LIN {X 0,Y 328.077,Z 664.549,A -85,B 0,C 180,E1 11851.958,E2 11851.958} C_VEL
LIN {X 0,Y 322.786,Z 698.857,A -85,B 0,C 180,E1 11850.839,E2 11850.839} C_VEL
LIN {X 0,Y 316.896,Z 730.284,A -85,B 0,C 180,E1 11849.561,E2 11849.561} C_VEL
LIN {X 0,Y 311.115,Z 757.419,A -85,B 0,C 180,E1 11848.161,E2 11848.161} C_VEL
LIN {X 0,Y 304.372,Z 786.191,A -85,B 0,C 180,E1 11846.363,E2 11846.363} C_VEL
LIN {X 0,Y 299.425,Z 805.619,A -85,B 0,C 180,E1 11844.9,E2 11844.9} C_VEL
LIN {X 0,Y 293.873,Z 823.687,A -85,B 0,C 180,E1 11843.236,E2 11843.236} C_VEL
LIN {X 0,Y 287.194,Z 842.545,A -85,B 0,C 180,E1 11841.082,E2 11841.082} C_VEL
LIN {X 0,Y 280.407,Z 859.77,A -85,B 0,C 180,E1 11838.643,E2 11838.643} C_VEL
LIN {X 0,Y 273.402,Z 876.134,A -85,B 0,C 180,E1 11835.792,E2 11835.792} C_VEL
LIN {X 0,Y 266.367,Z 891.442,A -85,B 0,C 180,E1 11832.507,E2 11832.507} C_VEL
LIN {X 0,Y 259.868,Z 905.271,A -85,B 0,C 180,E1 11828.842,E2 11828.842} C_VEL
LIN {X 0,Y 253.731,Z 918.322,A -85,B 0,C 180,E1 11824.574,E2 11824.574} C_VEL
LIN {X 0,Y 248.904,Z 929.249,A -85,B 0,C 180,E1 11820.142,E2 11820.142} C_VEL
LIN {X 0,Y 245.191,Z 938.697,A -85,B 0,C 180,E1 11815.353,E2 11815.353} C_VEL
LIN {X 0,Y 242.779,Z 946.583,A -85,B 0,C 180,E1 11810.24,E2 11810.24} C_VEL
LIN {X 0,Y 241.703,Z 952.882,A -85,B 0,C 180,E1 11804.861,E2 11804.861} C_VEL
LIN {X 0,Y 241.721,Z 956.944,A -85,B 0,C 180,E1 11800.005,E2 11800.005} C_VEL
LIN {X 0,Y 242.274,Z 959.368,A -85,B 0,C 180,E1 11795.447,E2 11795.447} C_VEL
LIN {X 0,Y 242.69,Z 960.344,A -85,B 0,C 180,E1 11791.416,E2 11791.416} C_VEL
LIN {X 0,Y 242.617,Z 960.808,A -85,B 0,C 180,E1 11788.347,E2 11788.347} C_VEL
LIN {X 0,Y 241.989,Z 961.423,A -85,B 0,C 180,E1 11784.309,E2 11784.309} C_VEL
LIN {X 0,Y 241.324,Z 960.912,A -85,B 0,C 180,E1 11779.737,E2 11779.737} C_VEL
LIN {X 0,Y 241.346,Z 959.091,A -85,B 0,C 180,E1 11774.624,E2 11774.624} C_VEL
LIN {X 0,Y 243.205,Z 954.97,A -85,B 0,C 180,E1 11768.029,E2 11768.029} C_VEL
LIN {X 0,Y 247.543,Z 949.265,A -85,B 0,C 180,E1 11761.71,E2 11761.71} C_VEL
LIN {X 0,Y 256.061,Z 940.692,A -85,B 0,C 180,E1 11754.695,E2 11754.695} C_VEL
LIN {X 0,Y 268.48,Z 930.238,A -85,B 0,C 180,E1 11748.191,E2 11748.191} C_VEL
LIN {X 0,Y 284.499,Z 918.06,A -85,B 0,C 180,E1 11742.434,E2 11742.434} C_VEL
LIN {X 0,Y 303.916,Z 904.379,A -85,B 0,C 180,E1 11737.492,E2 11737.492} C_VEL
LIN {X 0,Y 306.388,Z 902.677,A -85,B 0,C 180,E1 11736.938,E2 11736.938} C_VEL
LIN {X 0,Y 290.077,Z 909.42,A -85,B 0,C 180,E1 11732.999,E2 11732.999} C_VEL
LIN {X 0,Y 276.681,Z 914.167,A -85,B 0,C 180,E1 11728.728,E2 11728.728} C_VEL
LIN {X 0,Y 266.306,Z 916.874,A -85,B 0,C 180,E1 11724.394,E2 11724.394} C_VEL
LIN {X 0,Y 258.186,Z 917.772,A -85,B 0,C 180,E1 11719.926,E2 11719.926} C_VEL
LIN {X 0,Y 251.859,Z 916.837,A -85,B 0,C 180,E1 11715.19,E2 11715.19} C_VEL
LIN {X 0,Y 247.469,Z 914.048,A -85,B 0,C 180,E1 11710.476,E2 11710.476} C_VEL
LIN {X 0,Y 244.669,Z 909.579,A -85,B 0,C 180,E1 11705.864,E2 11705.864} C_VEL
LIN {X 0,Y 243.134,Z 903.597,A -85,B 0,C 180,E1 11701.414,E2 11701.414} C_VEL
LIN {X 0,Y 242.48,Z 895.781,A -85,B 0,C 180,E1 11696.927,E2 11696.927} C_VEL
LIN {X 0,Y 242.581,Z 886.484,A -85,B 0,C 180,E1 11692.659,E2 11692.659} C_VEL
LIN {X 0,Y 243.385,Z 875.099,A -85,B 0,C 180,E1 11688.387,E2 11688.387} C_VEL
LIN {X 0,Y 244.879,Z 862.174,A -85,B 0,C 180,E1 11684.366,E2 11684.366} C_VEL
LIN {X 0,Y 247.165,Z 846.76,A -85,B 0,C 180,E1 11680.38,E2 11680.38} C_VEL
LIN {X 0,Y 250.095,Z 829.651,A -85,B 0,C 180,E1 11676.684,E2 11676.684} C_VEL
LIN {X 0,Y 253.558,Z 810.82,A -85,B 0,C 180,E1 11673.285,E2 11673.285} C_VEL
LIN {X 0,Y 256.349,Z 796.184,A -85,B 0,C 180,E1 11671.015,E2 11671.015} C_VEL
LIN {X 0,Y 258.063,Z 795.879,A -85,B 0,C 180,E1 11670.267,E2 11670.267} C_VEL
LIN {X 0,Y 261.396,Z 793.79,A -85,B 0,C 180,E1 11669.419,E2 11669.419} C_VEL
LIN {X 0,Y 263.426,Z 792.151,A -85,B 0,C 180,E1 11669.048,E2 11669.048} C_VEL
LIN {X 0,Y 266.688,Z 790.708,A -85,B 0,C 180,E1 11668.085,E2 11668.085} C_VEL
LIN {X 0,Y 271.264,Z 787.43,A -85,B 0,C 180,E1 11667.19,E2 11667.19} C_VEL
LIN {X 0,Y 272.706,Z 786.509,A -85,B 0,C 180,E1 11666.885,E2 11666.885} C_VEL
LIN {X 0,Y 276.903,Z 784.082,A -85,B 0,C 180,E1 11665.965,E2 11665.965} C_VEL
LIN {X 0,Y 281.977,Z 780.134,A -85,B 0,C 180,E1 11665.186,E2 11665.186} C_VEL
LIN {X 0,Y 287.29,Z 776.786,A -85,B 0,C 180,E1 11664.188,E2 11664.188} C_VEL
LIN {X 0,Y 294.134,Z 771.195,A -85,B 0,C 180,E1 11663.251,E2 11663.251} C_VEL
LIN {X 0,Y 300.69,Z 766.466,A -85,B 0,C 180,E1 11662.276,E2 11662.276} C_VEL
LIN {X 0,Y 308.157,Z 759.605,A -85,B 0,C 180,E1 11661.465,E2 11661.465} C_VEL
LIN {X 0,Y 313.629,Z 755.169,A -85,B 0,C 180,E1 11660.78,E2 11660.78} C_VEL
LIN {X 0,Y 307.091,Z 774.598,A -85,B 0,C 180,E1 11658.904,E2 11658.904} C_VEL
LIN {X 0,Y 299.717,Z 793.413,A -85,B 0,C 180,E1 11656.659,E2 11656.659} C_VEL
LIN {X 0,Y 292.142,Z 810.488,A -85,B 0,C 180,E1 11654.147,E2 11654.147} C_VEL
LIN {X 0,Y 284.54,Z 825.999,A -85,B 0,C 180,E1 11651.349,E2 11651.349} C_VEL
LIN {X 0,Y 276.841,Z 840.469,A -85,B 0,C 180,E1 11648.142,E2 11648.142} C_VEL
LIN {X 0,Y 269.273,Z 853.798,A -85,B 0,C 180,E1 11644.477,E2 11644.477} C_VEL
LIN {X 0,Y 262.342,Z 865.452,A -85,B 0,C 180,E1 11640.459,E2 11640.459} C_VEL
LIN {X 0,Y 256.338,Z 875.316,A -85,B 0,C 180,E1 11636.154,E2 11636.154} C_VEL
LIN {X 0,Y 251.296,Z 883.626,A -85,B 0,C 180,E1 11631.473,E2 11631.473} C_VEL
LIN {X 0,Y 247.54,Z 890.026,A -85,B 0,C 180,E1 11626.666,E2 11626.666} C_VEL
LIN {X 0,Y 244.982,Z 894.672,A -85,B 0,C 180,E1 11621.775,E2 11621.775} C_VEL
LIN {X 0,Y 243.461,Z 897.762,A -85,B 0,C 180,E1 11616.604,E2 11616.604} C_VEL
LIN {X 0,Y 242.869,Z 899.092,A -85,B 0,C 180,E1 11611.652,E2 11611.652} C_VEL
LIN {X 0,Y 242.961,Z 898.929,A -85,B 0,C 180,E1 11606.933,E2 11606.933} C_VEL
LIN {X 0,Y 243.762,Z 897.219,A -85,B 0,C 180,E1 11601.983,E2 11601.983} C_VEL
LIN {X 0,Y 245.567,Z 893.689,A -85,B 0,C 180,E1 11596.82,E2 11596.82} C_VEL
LIN {X 0,Y 248.612,Z 888.313,A -85,B 0,C 180,E1 11591.717,E2 11591.717} C_VEL
LIN {X 0,Y 252.766,Z 881.335,A -85,B 0,C 180,E1 11586.945,E2 11586.945} C_VEL
LIN {X 0,Y 258.227,Z 872.413,A -85,B 0,C 180,E1 11582.312,E2 11582.312} C_VEL
LIN {X 0,Y 264.619,Z 861.893,A -85,B 0,C 180,E1 11578.062,E2 11578.062} C_VEL
LIN {X 0,Y 271.738,Z 849.807,A -85,B 0,C 180,E1 11574.193,E2 11574.193} C_VEL
LIN {X 0,Y 279.361,Z 836.154,A -85,B 0,C 180,E1 11570.69,E2 11570.69} C_VEL
LIN {X 0,Y 287.198,Z 821.088,A -85,B 0,C 180,E1 11567.569,E2 11567.569} C_VEL
LIN {X 0,Y 294.856,Z 804.991,A -85,B 0,C 180,E1 11564.858,E2 11564.858} C_VEL
LIN {X 0,Y 302.293,Z 787.594,A -85,B 0,C 180,E1 11562.472,E2 11562.472} C_VEL
LIN {X 0,Y 308.95,Z 769.937,A -85,B 0,C 180,E1 11560.487,E2 11560.487} C_VEL
LIN {X 0,Y 314.933,Z 751.546,A -85,B 0,C 180,E1 11558.79,E2 11558.79} C_VEL
LIN {X 0,Y 320.446,Z 731.196,A -85,B 0,C 180,E1 11557.281,E2 11557.281} C_VEL
LIN {X 0,Y 324.897,Z 710.419,A -85,B 0,C 180,E1 11556.057,E2 11556.057} C_VEL
LIN {X 0,Y 331.323,Z 672.15,A -85,B 0,C 180,E1 11554.363,E2 11554.363} C_VEL
LIN {X 0,Y 337.946,Z 631.963,A -85,B 0,C 180,E1 11552.979,E2 11552.979} C_VEL
LIN {X 0,Y 345.288,Z 583.472,A -85,B 0,C 180,E1 11551.669,E2 11551.669} C_VEL
LIN {X 0,Y 346.837,Z 571.682,A -85,B 0,C 180,E1 11551.387,E2 11551.387} C_VEL
LIN {X 0,Y 347.343,Z 564.173,A -85,B 0,C 180,E1 11551.067,E2 11551.067} C_VEL
LIN {X 0,Y 346.659,Z 544.539,A -85,B 0,C 180,E1 11549.728,E2 11549.728} C_VEL
LIN {X 0,Y 346.997,Z 538.052,A -85,B 0,C 180,E1 11549.49,E2 11549.49} C_VEL
LIN {X 0,Y 352.357,Z 479.815,A -85,B 0,C 180,E1 11548.405,E2 11548.405} C_VEL
LIN {X 0,Y 354.602,Z 455.735,A -85,B 0,C 180,E1 11547.969,E2 11547.969} C_VEL
LIN {X 0,Y 359.756,Z 433.802,A -85,B 0,C 180,E1 11547.297,E2 11547.297} C_VEL
LIN {X 0,Y 355.977,Z 420.386,A -85,B 0,C 180,E1 11544.167,E2 11544.167} C_VEL
LIN {X 0,Y 352.347,Z 408.944,A -85,B 0,C 180,E1 11540.951,E2 11540.951} C_VEL
LIN {X 0,Y 349.186,Z 399.554,A -85,B 0,C 180,E1 11537.756,E2 11537.756} C_VEL
LIN {X 0,Y 346.458,Z 391.969,A -85,B 0,C 180,E1 11534.542,E2 11534.542} C_VEL
LIN {X 0,Y 344.769,Z 387.315,A -85,B 0,C 180,E1 11532.138,E2 11532.138} C_VEL
LIN {X 0,Y 343.643,Z 384.271,A -85,B 0,C 180,E1 11530.308,E2 11530.308} C_VEL
LIN {X 0,Y 342.522,Z 380.827,A -85,B 0,C 180,E1 11527.886,E2 11527.886} C_VEL
LIN {X 0,Y 341.574,Z 376.877,A -85,B 0,C 180,E1 11524.113,E2 11524.113} C_VEL
LIN {X 0,Y 341.688,Z 375.496,A -85,B 0,C 180,E1 11518.323,E2 11518.323} C_VEL
LIN {X 0,Y 343.463,Z 376.678,A -85,B 0,C 180,E1 11513.691,E2 11513.691} C_VEL
LIN {X 0,Y 344.276,Z 386.078,A -85,B 0,C 180,E1 11510.429,E2 11510.429} C_VEL
LIN {X 0,Y 345.899,Z 396.844,A -85,B 0,C 180,E1 11507.097,E2 11507.097} C_VEL
LIN {X 0,Y 350.144,Z 415.442,A -85,B 0,C 180,E1 11502.208,E2 11502.208} C_VEL
LIN {X 0,Y 352.332,Z 423.731,A -85,B 0,C 180,E1 11500.349,E2 11500.349} C_VEL
LIN {X 0,Y 353.872,Z 430.799,A -85,B 0,C 180,E1 11499.043,E2 11499.043} C_VEL
LIN {X 0,Y 333.513,Z 567.002,A -85,B 0,C 180,E1 11495.422,E2 11495.422} C_VEL
LIN {X 0,Y 328.621,Z 627.947,A -85,B 0,C 180,E1 11494.129,E2 11494.129} C_VEL
LIN {X 0,Y 324.389,Z 662.655,A -85,B 0,C 180,E1 11493.239,E2 11493.239} C_VEL
LIN {X 0,Y 319.068,Z 696.214,A -85,B 0,C 180,E1 11492.157,E2 11492.157} C_VEL
LIN {X 0,Y 313.154,Z 727.135,A -85,B 0,C 180,E1 11490.935,E2 11490.935} C_VEL
LIN {X 0,Y 306.952,Z 755.501,A -85,B 0,C 180,E1 11489.497,E2 11489.497} C_VEL
LIN {X 0,Y 299.604,Z 786.015,A -85,B 0,C 180,E1 11487.603,E2 11487.603} C_VEL
LIN {X 0,Y 293.809,Z 807.39,A -85,B 0,C 180,E1 11485.963,E2 11485.963} C_VEL
LIN {X 0,Y 287.815,Z 825.742,A -85,B 0,C 180,E1 11484.213,E2 11484.213} C_VEL
LIN {X 0,Y 280.907,Z 844.161,A -85,B 0,C 180,E1 11482.039,E2 11482.039} C_VEL
LIN {X 0,Y 273.611,Z 861.525,A -85,B 0,C 180,E1 11479.475,E2 11479.475} C_VEL
LIN {X 0,Y 266.144,Z 877.913,A -85,B 0,C 180,E1 11476.476,E2 11476.476} C_VEL
LIN {X 0,Y 258.919,Z 892.811,A -85,B 0,C 180,E1 11473.121,E2 11473.121} C_VEL
LIN {X 0,Y 252.232,Z 906.31,A -85,B 0,C 180,E1 11469.365,E2 11469.365} C_VEL
LIN {X 0,Y 246.224,Z 918.438,A -85,B 0,C 180,E1 11465.215,E2 11465.215} C_VEL
LIN {X 0,Y 241.198,Z 929.146,A -85,B 0,C 180,E1 11460.657,E2 11460.657} C_VEL
LIN {X 0,Y 237.18,Z 938.805,A -85,B 0,C 180,E1 11455.468,E2 11455.468} C_VEL
LIN {X 0,Y 234.746,Z 946.482,A -85,B 0,C 180,E1 11450.183,E2 11450.183} C_VEL
LIN {X 0,Y 233.715,Z 952.415,A -85,B 0,C 180,E1 11444.785,E2 11444.785} C_VEL
LIN {X 0,Y 233.795,Z 956.418,A -85,B 0,C 180,E1 11439.601,E2 11439.601} C_VEL
LIN {X 0,Y 234.399,Z 958.644,A -85,B 0,C 180,E1 11434.894,E2 11434.894} C_VEL
LIN {X 0,Y 234.776,Z 959.382,A -85,B 0,C 180,E1 11430.976,E2 11430.976} C_VEL
LIN {X 0,Y 234.655,Z 959.491,A -85,B 0,C 180,E1 11427.558,E2 11427.558} C_VEL
LIN {X 0,Y 233.929,Z 960.029,A -85,B 0,C 180,E1 11423.373,E2 11423.373} C_VEL
LIN {X 0,Y 233.324,Z 959.466,A -85,B 0,C 180,E1 11418.631,E2 11418.631} C_VEL
LIN {X 0,Y 233.566,Z 957.616,A -85,B 0,C 180,E1 11413.332,E2 11413.332} C_VEL
LIN {X 0,Y 236.074,Z 953.379,A -85,B 0,C 180,E1 11406.273,E2 11406.273} C_VEL
LIN {X 0,Y 241.373,Z 947.552,A -85,B 0,C 180,E1 11399.643,E2 11399.643} C_VEL
LIN {X 0,Y 251.549,Z 938.733,A -85,B 0,C 180,E1 11392.255,E2 11392.255} C_VEL
LIN {X 0,Y 265.876,Z 928.157,A -85,B 0,C 180,E1 11385.613,E2 11385.613} C_VEL
LIN {X 0,Y 283.382,Z 916.29,A -85,B 0,C 180,E1 11380.033,E2 11380.033} C_VEL
LIN {X 0,Y 296.308,Z 907.981,A -85,B 0,C 180,E1 11376.863,E2 11376.863} C_VEL
LIN {X 0,Y 280.326,Z 913.596,A -85,B 0,C 180,E1 11372.831,E2 11372.831} C_VEL
LIN {X 0,Y 267.516,Z 917.249,A -85,B 0,C 180,E1 11368.583,E2 11368.583} C_VEL
LIN {X 0,Y 257.188,Z 919.111,A -85,B 0,C 180,E1 11364.093,E2 11364.093} C_VEL
LIN {X 0,Y 248.834,Z 919.122,A -85,B 0,C 180,E1 11359.239,E2 11359.239} C_VEL
LIN {X 0,Y 242.975,Z 917.338,A -85,B 0,C 180,E1 11354.538,E2 11354.538} C_VEL
LIN {X 0,Y 238.945,Z 913.958,A -85,B 0,C 180,E1 11349.879,E2 11349.879} C_VEL
LIN {X 0,Y 236.299,Z 908.835,A -85,B 0,C 180,E1 11345.098,E2 11345.098} C_VEL
LIN {X 0,Y 234.928,Z 902.216,A -85,B 0,C 180,E1 11340.488,E2 11340.488} C_VEL
LIN {X 0,Y 234.446,Z 894.223,A -85,B 0,C 180,E1 11336.087,E2 11336.087} C_VEL
LIN {X 0,Y 234.7,Z 884.316,A -85,B 0,C 180,E1 11331.671,E2 11331.671} C_VEL
LIN {X 0,Y 235.701,Z 872.242,A -85,B 0,C 180,E1 11327.256,E2 11327.256} C_VEL
LIN {X 0,Y 237.448,Z 858.577,A -85,B 0,C 180,E1 11323.108,E2 11323.108} C_VEL
LIN {X 0,Y 239.856,Z 843.366,A -85,B 0,C 180,E1 11319.247,E2 11319.247} C_VEL
LIN {X 0,Y 242.896,Z 826.279,A -85,B 0,C 180,E1 11315.618,E2 11315.618} C_VEL
LIN {X 0,Y 246.544,Z 807.022,A -85,B 0,C 180,E1 11312.199,E2 11312.199} C_VEL
LIN {X 0,Y 246.823,Z 806.063,A -85,B 0,C 180,E1 11311.971,E2 11311.971} C_VEL
LIN {X 0,Y 248.589,Z 805.719,A -85,B 0,C 180,E1 11311.14,E2 11311.14} C_VEL
LIN {X 0,Y 251.85,Z 803.755,A -85,B 0,C 180,E1 11310.246,E2 11310.246} C_VEL
LIN {X 0,Y 253.415,Z 802.585,A -85,B 0,C 180,E1 11309.927,E2 11309.927} C_VEL
LIN {X 0,Y 256.887,Z 801.096,A -85,B 0,C 180,E1 11308.823,E2 11308.823} C_VEL
LIN {X 0,Y 261.355,Z 798.141,A -85,B 0,C 180,E1 11307.874,E2 11307.874} C_VEL
LIN {X 0,Y 265.965,Z 795.781,A -85,B 0,C 180,E1 11306.709,E2 11306.709} C_VEL
LIN {X 0,Y 270.732,Z 792.531,A -85,B 0,C 180,E1 11305.849,E2 11305.849} C_VEL
LIN {X 0,Y 275.815,Z 789.679,A -85,B 0,C 180,E1 11304.801,E2 11304.801} C_VEL
LIN {X 0,Y 281.675,Z 785.442,A -85,B 0,C 180,E1 11303.895,E2 11303.895} C_VEL
LIN {X 0,Y 288.032,Z 781.326,A -85,B 0,C 180,E1 11302.84,E2 11302.84} C_VEL
LIN {X 0,Y 294.281,Z 776.492,A -85,B 0,C 180,E1 11302.049,E2 11302.049} C_VEL
LIN {X 0,Y 301.059,Z 771.653,A -85,B 0,C 180,E1 11301.118,E2 11301.118} C_VEL
LIN {X 0,Y 304.437,Z 768.801,A -85,B 0,C 180,E1 11300.753,E2 11300.753} C_VEL
LIN {X 0,Y 297.401,Z 787.222,A -85,B 0,C 180,E1 11298.714,E2 11298.714} C_VEL
LIN {X 0,Y 289.716,Z 804.818,A -85,B 0,C 180,E1 11296.321,E2 11296.321} C_VEL
LIN {X 0,Y 281.607,Z 821.407,A -85,B 0,C 180,E1 11293.538,E2 11293.538} C_VEL
LIN {X 0,Y 273.828,Z 835.892,A -85,B 0,C 180,E1 11290.54,E2 11290.54} C_VEL
LIN {X 0,Y 266.256,Z 849.006,A -85,B 0,C 180,E1 11287.201,E2 11287.201} C_VEL
LIN {X 0,Y 259.078,Z 860.781,A -85,B 0,C 180,E1 11283.497,E2 11283.497} C_VEL
LIN {X 0,Y 252.194,Z 871.677,A -85,B 0,C 180,E1 11279.188,E2 11279.188} C_VEL
LIN {X 0,Y 246.468,Z 880.603,A -85,B 0,C 180,E1 11274.667,E2 11274.667} C_VEL
LIN {X 0,Y 241.823,Z 887.928,A -85,B 0,C 180,E1 11269.819,E2 11269.819} C_VEL
LIN {X 0,Y 238.462,Z 893.471,A -85,B 0,C 180,E1 11264.82,E2 11264.82} C_VEL
LIN {X 0,Y 236.24,Z 897.45,A -85,B 0,C 180,E1 11259.501,E2 11259.501} C_VEL
LIN {X 0,Y 235.164,Z 899.596,A -85,B 0,C 180,E1 11254.39,E2 11254.39} C_VEL
LIN {X 0,Y 234.899,Z 900.206,A -85,B 0,C 180,E1 11249.512,E2 11249.512} C_VEL
LIN {X 0,Y 235.336,Z 899.324,A -85,B 0,C 180,E1 11244.392,E2 11244.392} C_VEL
LIN {X 0,Y 236.607,Z 896.831,A -85,B 0,C 180,E1 11239.284,E2 11239.284} C_VEL
LIN {X 0,Y 238.961,Z 892.703,A -85,B 0,C 180,E1 11234.218,E2 11234.218} C_VEL
LIN {X 0,Y 242.348,Z 887.166,A -85,B 0,C 180,E1 11229.47,E2 11229.47} C_VEL
LIN {X 0,Y 246.933,Z 879.968,A -85,B 0,C 180,E1 11224.839,E2 11224.839} C_VEL
LIN {X 0,Y 252.733,Z 870.958,A -85,B 0,C 180,E1 11220.361,E2 11220.361} C_VEL
LIN {X 0,Y 259.345,Z 860.52,A -85,B 0,C 180,E1 11216.277,E2 11216.277} C_VEL
LIN {X 0,Y 266.99,Z 847.977,A -85,B 0,C 180,E1 11212.379,E2 11212.379} C_VEL
LIN {X 0,Y 274.638,Z 834.658,A -85,B 0,C 180,E1 11209.055,E2 11209.055} C_VEL
LIN {X 0,Y 282.74,Z 819.433,A -85,B 0,C 180,E1 11205.98,E2 11205.98} C_VEL
LIN {X 0,Y 290.627,Z 803.132,A -85,B 0,C 180,E1 11203.31,E2 11203.31} C_VEL
LIN {X 0,Y 298.105,Z 785.857,A -85,B 0,C 180,E1 11201.002,E2 11201.002} C_VEL
LIN {X 0,Y 305.095,Z 767.411,A -85,B 0,C 180,E1 11198.995,E2 11198.995} C_VEL
LIN {X 0,Y 311.158,Z 748.674,A -85,B 0,C 180,E1 11197.335,E2 11197.335} C_VEL
LIN {X 0,Y 316.591,Z 728.432,A -85,B 0,C 180,E1 11195.894,E2 11195.894} C_VEL
LIN {X 0,Y 320.965,Z 707.582,A -85,B 0,C 180,E1 11194.718,E2 11194.718} C_VEL
LIN {X 0,Y 327.652,Z 668.819,A -85,B 0,C 180,E1 11193.043,E2 11193.043} C_VEL
LIN {X 0,Y 334.631,Z 627.548,A -85,B 0,C 180,E1 11191.666,E2 11191.666} C_VEL
LIN {X 0,Y 341.901,Z 579.415,A -85,B 0,C 180,E1 11190.407,E2 11190.407} C_VEL
LIN {X 0,Y 346.997,Z 538.052,A -85,B 0,C 180,E1 11189.49,E2 11189.49} C_VEL
LIN {X 0,Y 347.349,Z 530.5,A -85,B 0,C 180,E1 11189.197,E2 11189.197} C_VEL
LIN {X 0,Y 346.384,Z 510.784,A -85,B 0,C 180,E1 11187.894,E2 11187.894} C_VEL
LIN {X 0,Y 346.622,Z 504.272,A -85,B 0,C 180,E1 11187.667,E2 11187.667} C_VEL
LIN {X 0,Y 350.786,Z 458.367,A -85,B 0,C 180,E1 11186.851,E2 11186.851} C_VEL
LIN {X 0,Y 355.639,Z 437.88,A -85,B 0,C 180,E1 11186.249,E2 11186.249} C_VEL
LIN {X 0,Y 352.368,Z 425.709,A -85,B 0,C 180,E1 11183.319,E2 11183.319} C_VEL
LIN {X 0,Y 349.155,Z 415.154,A -85,B 0,C 180,E1 11180.274,E2 11180.274} C_VEL
LIN {X 0,Y 346.39,Z 406.434,A -85,B 0,C 180,E1 11177.254,E2 11177.254} C_VEL
LIN {X 0,Y 343.844,Z 398.992,A -85,B 0,C 180,E1 11174.053,E2 11174.053} C_VEL
LIN {X 0,Y 342.325,Z 394.25,A -85,B 0,C 180,E1 11171.542,E2 11171.542} C_VEL
LIN {X 0,Y 341.3,Z 391.444,A -85,B 0,C 180,E1 11169.783,E2 11169.783} C_VEL
LIN {X 0,Y 340.4,Z 388.391,A -85,B 0,C 180,E1 11167.596,E2 11167.596} C_VEL
LIN {X 0,Y 339.526,Z 384.355,A -85,B 0,C 180,E1 11163.546,E2 11163.546} C_VEL
LIN {X 0,Y 339.949,Z 383.311,A -85,B 0,C 180,E1 11157.977,E2 11157.977} C_VEL
LIN {X 0,Y 341.472,Z 384.468,A -85,B 0,C 180,E1 11153.949,E2 11153.949} C_VEL
LIN {X 0,Y 342.19,Z 394.107,A -85,B 0,C 180,E1 11150.624,E2 11150.624} C_VEL
LIN {X 0,Y 343.611,Z 403.92,A -85,B 0,C 180,E1 11147.607,E2 11147.607} C_VEL
LIN {X 0,Y 347.54,Z 422.084,A -85,B 0,C 180,E1 11142.805,E2 11142.805} C_VEL
LIN {X 0,Y 349.46,Z 429.852,A -85,B 0,C 180,E1 11141.049,E2 11141.049} C_VEL
LIN {X 0,Y 350.422,Z 434.607,A -85,B 0,C 180,E1 11140.171,E2 11140.171} C_VEL
LIN {X 0,Y 330.399,Z 563.948,A -85,B 0,C 180,E1 11136.746,E2 11136.746} C_VEL
LIN {X 0,Y 325.235,Z 626.022,A -85,B 0,C 180,E1 11135.427,E2 11135.427} C_VEL
LIN {X 0,Y 320.852,Z 660.895,A -85,B 0,C 180,E1 11134.545,E2 11134.545} C_VEL
LIN {X 0,Y 315.405,Z 694.246,A -85,B 0,C 180,E1 11133.482,E2 11133.482} C_VEL
LIN {X 0,Y 309.434,Z 724.747,A -85,B 0,C 180,E1 11132.299,E2 11132.299} C_VEL
LIN {X 0,Y 302.933,Z 753.57,A -85,B 0,C 180,E1 11130.864,E2 11130.864} C_VEL
LIN {X 0,Y 295.72,Z 782.923,A -85,B 0,C 180,E1 11129.073,E2 11129.073} C_VEL
LIN {X 0,Y 290.179,Z 803.022,A -85,B 0,C 180,E1 11127.588,E2 11127.588} C_VEL
LIN {X 0,Y 283.713,Z 822.483,A -85,B 0,C 180,E1 11125.792,E2 11125.792} C_VEL
LIN {X 0,Y 276.538,Z 841.161,A -85,B 0,C 180,E1 11123.631,E2 11123.631} C_VEL
LIN {X 0,Y 268.902,Z 858.867,A -85,B 0,C 180,E1 11121.067,E2 11121.067} C_VEL
LIN {X 0,Y 261.419,Z 874.651,A -85,B 0,C 180,E1 11118.232,E2 11118.232} C_VEL
LIN {X 0,Y 253.722,Z 889.849,A -85,B 0,C 180,E1 11114.863,E2 11114.863} C_VEL
LIN {X 0,Y 246.148,Z 904.381,A -85,B 0,C 180,E1 11110.844,E2 11110.844} C_VEL
LIN {X 0,Y 239.379,Z 917.279,A -85,B 0,C 180,E1 11106.38,E2 11106.38} C_VEL
LIN {X 0,Y 233.997,Z 927.995,A -85,B 0,C 180,E1 11101.708,E2 11101.708} C_VEL
LIN {X 0,Y 229.81,Z 937.272,A -85,B 0,C 180,E1 11096.625,E2 11096.625} C_VEL
LIN {X 0,Y 226.972,Z 945.352,A -85,B 0,C 180,E1 11090.943,E2 11090.943} C_VEL
LIN {X 0,Y 225.786,Z 951.275,A -85,B 0,C 180,E1 11085.409,E2 11085.409} C_VEL
LIN {X 0,Y 225.772,Z 955.227,A -85,B 0,C 180,E1 11080.204,E2 11080.204} C_VEL
LIN {X 0,Y 226.384,Z 957.536,A -85,B 0,C 180,E1 11075.322,E2 11075.322} C_VEL
LIN {X 0,Y 226.821,Z 958.36,A -85,B 0,C 180,E1 11071.263,E2 11071.263} C_VEL
LIN {X 0,Y 226.729,Z 958.185,A -85,B 0,C 180,E1 11067.219,E2 11067.219} C_VEL
LIN {X 0,Y 225.883,Z 958.597,A -85,B 0,C 180,E1 11062.369,E2 11062.369} C_VEL
LIN {X 0,Y 225.37,Z 957.858,A -85,B 0,C 180,E1 11056.922,E2 11056.922} C_VEL
LIN {X 0,Y 226.13,Z 955.663,A -85,B 0,C 180,E1 11050.9,E2 11050.9} C_VEL
LIN {X 0,Y 229.876,Z 951.018,A -85,B 0,C 180,E1 11043.383,E2 11043.383} C_VEL
LIN {X 0,Y 237.165,Z 944.592,A -85,B 0,C 180,E1 11036.156,E2 11036.156} C_VEL
LIN {X 0,Y 249.299,Z 935.661,A -85,B 0,C 180,E1 11028.869,E2 11028.869} C_VEL
LIN {X 0,Y 266.188,Z 924.791,A -85,B 0,C 180,E1 11022.252,E2 11022.252} C_VEL
LIN {X 0,Y 286.276,Z 912.738,A -85,B 0,C 180,E1 11016.812,E2 11016.812} C_VEL
LIN {X 0,Y 271.104,Z 917.186,A -85,B 0,C 180,E1 11012.832,E2 11012.832} C_VEL
LIN {X 0,Y 257.814,Z 920.039,A -85,B 0,C 180,E1 11008.24,E2 11008.24} C_VEL
LIN {X 0,Y 247.222,Z 920.953,A -85,B 0,C 180,E1 11003.351,E2 11003.351} C_VEL
LIN {X 0,Y 239.471,Z 919.991,A -85,B 0,C 180,E1 10998.502,E2 10998.502} C_VEL
LIN {X 0,Y 233.867,Z 917.343,A -85,B 0,C 180,E1 10993.601,E2 10993.601} C_VEL
LIN {X 0,Y 229.964,Z 912.881,A -85,B 0,C 180,E1 10988.501,E2 10988.501} C_VEL
LIN {X 0,Y 227.69,Z 906.798,A -85,B 0,C 180,E1 10983.525,E2 10983.525} C_VEL
LIN {X 0,Y 226.676,Z 899.674,A -85,B 0,C 180,E1 10978.989,E2 10978.989} C_VEL
LIN {X 0,Y 226.455,Z 890.778,A -85,B 0,C 180,E1 10974.426,E2 10974.426} C_VEL
LIN {X 0,Y 227.003,Z 879.855,A -85,B 0,C 180,E1 10969.852,E2 10969.852} C_VEL
LIN {X 0,Y 228.331,Z 867.078,A -85,B 0,C 180,E1 10965.418,E2 10965.418} C_VEL
LIN {X 0,Y 230.407,Z 852.761,A -85,B 0,C 180,E1 10961.268,E2 10961.268} C_VEL
LIN {X 0,Y 233.226,Z 836.41,A -85,B 0,C 180,E1 10957.303,E2 10957.303} C_VEL
LIN {X 0,Y 236.629,Z 818.334,A -85,B 0,C 180,E1 10953.661,E2 10953.661} C_VEL
LIN {X 0,Y 237.276,Z 815.294,A -85,B 0,C 180,E1 10953.063,E2 10953.063} C_VEL
LIN {X 0,Y 239.193,Z 814.88,A -85,B 0,C 180,E1 10952.083,E2 10952.083} C_VEL
LIN {X 0,Y 242.409,Z 812.984,A -85,B 0,C 180,E1 10951.144,E2 10951.144} C_VEL
LIN {X 0,Y 243.699,Z 812.239,A -85,B 0,C 180,E1 10950.774,E2 10950.774} C_VEL
LIN {X 0,Y 247.112,Z 810.774,A -85,B 0,C 180,E1 10949.616,E2 10949.616} C_VEL
LIN {X 0,Y 250.748,Z 808.509,A -85,B 0,C 180,E1 10948.775,E2 10948.775} C_VEL
LIN {X 0,Y 255.175,Z 806.438,A -85,B 0,C 180,E1 10947.532,E2 10947.532} C_VEL
LIN {X 0,Y 259.649,Z 803.739,A -85,B 0,C 180,E1 10946.586,E2 10946.586} C_VEL
LIN {X 0,Y 264.64,Z 801.14,A -85,B 0,C 180,E1 10945.454,E2 10945.454} C_VEL
LIN {X 0,Y 269.4,Z 798.093,A -85,B 0,C 180,E1 10944.619,E2 10944.619} C_VEL
LIN {X 0,Y 275.506,Z 794.582,A -85,B 0,C 180,E1 10943.473,E2 10943.473} C_VEL
LIN {X 0,Y 281.455,Z 790.564,A -85,B 0,C 180,E1 10942.591,E2 10942.591} C_VEL
LIN {X 0,Y 288.642,Z 785.947,A -85,B 0,C 180,E1 10941.526,E2 10941.526} C_VEL
LIN {X 0,Y 294.44,Z 781.641,A -85,B 0,C 180,E1 10940.829,E2 10940.829} C_VEL
LIN {X 0,Y 295.133,Z 781.191,A -85,B 0,C 180,E1 10940.731,E2 10940.731} C_VEL
LIN {X 0,Y 287.625,Z 798.765,A -85,B 0,C 180,E1 10938.518,E2 10938.518} C_VEL
LIN {X 0,Y 279.607,Z 815.369,A -85,B 0,C 180,E1 10935.955,E2 10935.955} C_VEL
LIN {X 0,Y 271.285,Z 830.931,A -85,B 0,C 180,E1 10932.99,E2 10932.99} C_VEL
LIN {X 0,Y 263.105,Z 844.964,A -85,B 0,C 180,E1 10929.677,E2 10929.677} C_VEL
LIN {X 0,Y 255.273,Z 857.536,A -85,B 0,C 180,E1 10925.983,E2 10925.983} C_VEL
LIN {X 0,Y 247.995,Z 868.647,A -85,B 0,C 180,E1 10921.883,E2 10921.883} C_VEL
LIN {X 0,Y 241.508,Z 878.284,A -85,B 0,C 180,E1 10917.359,E2 10917.359} C_VEL
LIN {X 0,Y 236.274,Z 886.036,A -85,B 0,C 180,E1 10912.65,E2 10912.65} C_VEL
LIN {X 0,Y 232.134,Z 892.334,A -85,B 0,C 180,E1 10907.549,E2 10907.549} C_VEL
LIN {X 0,Y 229.303,Z 896.881,A -85,B 0,C 180,E1 10902.338,E2 10902.338} C_VEL
LIN {X 0,Y 227.654,Z 899.817,A -85,B 0,C 180,E1 10896.96,E2 10896.96} C_VEL
LIN {X 0,Y 226.989,Z 901.115,A -85,B 0,C 180,E1 10891.515,E2 10891.515} C_VEL
LIN {X 0,Y 227.125,Z 900.87,A -85,B 0,C 180,E1 10886.467,E2 10886.467} C_VEL
LIN {X 0,Y 228.019,Z 899.232,A -85,B 0,C 180,E1 10881.426,E2 10881.426} C_VEL
LIN {X 0,Y 230.071,Z 895.719,A -85,B 0,C 180,E1 10875.914,E2 10875.914} C_VEL
LIN {X 0,Y 233.499,Z 890.361,A -85,B 0,C 180,E1 10870.488,E2 10870.488} C_VEL
LIN {X 0,Y 238.149,Z 883.406,A -85,B 0,C 180,E1 10865.439,E2 10865.439} C_VEL
LIN {X 0,Y 244.19,Z 874.496,A -85,B 0,C 180,E1 10860.57,E2 10860.57} C_VEL
LIN {X 0,Y 251.207,Z 863.989,A -85,B 0,C 180,E1 10856.135,E2 10856.135} C_VEL
LIN {X 0,Y 258.967,Z 851.916,A -85,B 0,C 180,E1 10852.127,E2 10852.127} C_VEL
LIN {X 0,Y 266.745,Z 839.131,A -85,B 0,C 180,E1 10848.721,E2 10848.721} C_VEL
LIN {X 0,Y 275.248,Z 824.016,A -85,B 0,C 180,E1 10845.484,E2 10845.484} C_VEL
LIN {X 0,Y 283.297,Z 808.339,A -85,B 0,C 180,E1 10842.766,E2 10842.766} C_VEL
LIN {X 0,Y 291.225,Z 791.102,A -85,B 0,C 180,E1 10840.34,E2 10840.34} C_VEL
LIN {X 0,Y 298.585,Z 772.846,A -85,B 0,C 180,E1 10838.253,E2 10838.253} C_VEL
LIN {X 0,Y 304.934,Z 754.573,A -85,B 0,C 180,E1 10836.548,E2 10836.548} C_VEL
LIN {X 0,Y 310.474,Z 735.613,A -85,B 0,C 180,E1 10835.114,E2 10835.114} C_VEL
LIN {X 0,Y 315.348,Z 714.589,A -85,B 0,C 180,E1 10833.846,E2 10833.846} C_VEL
LIN {X 0,Y 321.971,Z 677.886,A -85,B 0,C 180,E1 10832.183,E2 10832.183} C_VEL
LIN {X 0,Y 328.782,Z 638.901,A -85,B 0,C 180,E1 10830.802,E2 10830.802} C_VEL
LIN {X 0,Y 336.281,Z 592.581,A -85,B 0,C 180,E1 10829.532,E2 10829.532} C_VEL
LIN {X 0,Y 342.481,Z 545.441,A -85,B 0,C 180,E1 10828.46,E2 10828.46} C_VEL
LIN {X 0,Y 346.622,Z 504.272,A -85,B 0,C 180,E1 10827.667,E2 10827.667} C_VEL
LIN {X 0,Y 346.827,Z 496.694,A -85,B 0,C 180,E1 10827.387,E2 10827.387} C_VEL
LIN {X 0,Y 345.781,Z 476.925,A -85,B 0,C 180,E1 10826.107,E2 10826.107} C_VEL
LIN {X 0,Y 346.043,Z 470.407,A -85,B 0,C 180,E1 10825.886,E2 10825.886} C_VEL
LIN {X 0,Y 347.16,Z 460.863,A -85,B 0,C 180,E1 10825.703,E2 10825.703} C_VEL
LIN {X 0,Y 351.671,Z 441.871,A -85,B 0,C 180,E1 10825.155,E2 10825.155} C_VEL
LIN {X 0,Y 348.557,Z 429.987,A -85,B 0,C 180,E1 10822.162,E2 10822.162} C_VEL
LIN {X 0,Y 345.457,Z 419.294,A -85,B 0,C 180,E1 10818.916,E2 10818.916} C_VEL
LIN {X 0,Y 342.728,Z 410.383,A -85,B 0,C 180,E1 10815.569,E2 10815.569} C_VEL
LIN {X 0,Y 340.438,Z 403.169,A -85,B 0,C 180,E1 10812.122,E2 10812.122} C_VEL
LIN {X 0,Y 339.23,Z 399.196,A -85,B 0,C 180,E1 10809.672,E2 10809.672} C_VEL
LIN {X 0,Y 338.271,Z 395.951,A -85,B 0,C 180,E1 10807.302,E2 10807.302} C_VEL
LIN {X 0,Y 337.59,Z 392.091,A -85,B 0,C 180,E1 10803.396,E2 10803.396} C_VEL
LIN {X 0,Y 338.009,Z 391.072,A -85,B 0,C 180,E1 10797.966,E2 10797.966} C_VEL
LIN {X 0,Y 339.487,Z 392.138,A -85,B 0,C 180,E1 10794.253,E2 10794.253} C_VEL
LIN {X 0,Y 340.126,Z 402.438,A -85,B 0,C 180,E1 10790.738,E2 10790.738} C_VEL
LIN {X 0,Y 341.317,Z 411.018,A -85,B 0,C 180,E1 10788.114,E2 10788.114} C_VEL
LIN {X 0,Y 344.996,Z 428.89,A -85,B 0,C 180,E1 10783.369,E2 10783.369} C_VEL
LIN {X 0,Y 346.692,Z 436.289,A -85,B 0,C 180,E1 10781.699,E2 10781.699} C_VEL
LIN {X 0,Y 347.021,Z 438.508,A -85,B 0,C 180,E1 10781.313,E2 10781.313} C_VEL
LIN {X 0,Y 327.455,Z 561.023,A -85,B 0,C 180,E1 10778.093,E2 10778.093} C_VEL
LIN {X 0,Y 322.042,Z 623.917,A -85,B 0,C 180,E1 10776.757,E2 10776.757} C_VEL
LIN {X 0,Y 317.459,Z 659.337,A -85,B 0,C 180,E1 10775.875,E2 10775.875} C_VEL
LIN {X 0,Y 311.746,Z 693.302,A -85,B 0,C 180,E1 10774.804,E2 10774.804} C_VEL
LIN {X 0,Y 304.7,Z 727.554,A -85,B 0,C 180,E1 10773.461,E2 10773.461} C_VEL
LIN {X 0,Y 297.83,Z 757.286,A -85,B 0,C 180,E1 10771.965,E2 10771.965} C_VEL
LIN {X 0,Y 289.758,Z 788.404,A -85,B 0,C 180,E1 10770.013,E2 10770.013} C_VEL
LIN {X 0,Y 283.881,Z 807.826,A -85,B 0,C 180,E1 10768.471,E2 10768.471} C_VEL
LIN {X 0,Y 277.441,Z 825.662,A -85,B 0,C 180,E1 10766.733,E2 10766.733} C_VEL
LIN {X 0,Y 269.721,Z 844.322,A -85,B 0,C 180,E1 10764.46,E2 10764.46} C_VEL
LIN {X 0,Y 261.879,Z 861.341,A -85,B 0,C 180,E1 10761.863,E2 10761.863} C_VEL
LIN {X 0,Y 253.797,Z 877.457,A -85,B 0,C 180,E1 10758.806,E2 10758.806} C_VEL
LIN {X 0,Y 245.707,Z 892.542,A -85,B 0,C 180,E1 10755.25,E2 10755.25} C_VEL
LIN {X 0,Y 238.201,Z 906.098,A -85,B 0,C 180,E1 10751.226,E2 10751.226} C_VEL
LIN {X 0,Y 231.304,Z 918.5,A -85,B 0,C 180,E1 10746.623,E2 10746.623} C_VEL
LIN {X 0,Y 225.602,Z 929.356,A -85,B 0,C 180,E1 10741.533,E2 10741.533} C_VEL
LIN {X 0,Y 221.317,Z 938.634,A -85,B 0,C 180,E1 10735.991,E2 10735.991} C_VEL
LIN {X 0,Y 218.761,Z 945.881,A -85,B 0,C 180,E1 10730.327,E2 10730.327} C_VEL
LIN {X 0,Y 217.751,Z 951.329,A -85,B 0,C 180,E1 10724.629,E2 10724.629} C_VEL
LIN {X 0,Y 217.911,Z 954.912,A -85,B 0,C 180,E1 10719.241,E2 10719.241} C_VEL
LIN {X 0,Y 218.581,Z 956.866,A -85,B 0,C 180,E1 10714.258,E2 10714.258} C_VEL
LIN {X 0,Y 218.913,Z 957.435,A -85,B 0,C 180,E1 10710.262,E2 10710.262} C_VEL
LIN {X 0,Y 218.663,Z 956.951,A -85,B 0,C 180,E1 10706.067,E2 10706.067} C_VEL
LIN {X 0,Y 217.776,Z 957.092,A -85,B 0,C 180,E1 10700.804,E2 10700.804} C_VEL
LIN {X 0,Y 217.499,Z 956.197,A -85,B 0,C 180,E1 10695.081,E2 10695.081} C_VEL
LIN {X 0,Y 218.932,Z 953.783,A -85,B 0,C 180,E1 10688.569,E2 10688.569} C_VEL
LIN {X 0,Y 223.988,Z 948.853,A -85,B 0,C 180,E1 10680.591,E2 10680.591} C_VEL
LIN {X 0,Y 233.054,Z 942.206,A -85,B 0,C 180,E1 10673.083,E2 10673.083} C_VEL
LIN {X 0,Y 247.522,Z 933.039,A -85,B 0,C 180,E1 10665.665,E2 10665.665} C_VEL
LIN {X 0,Y 266.25,Z 922.437,A -85,B 0,C 180,E1 10659.319,E2 10659.319} C_VEL
LIN {X 0,Y 276.164,Z 917.011,A -85,B 0,C 180,E1 10656.756,E2 10656.756} C_VEL
LIN {X 0,Y 260.678,Z 920.591,A -85,B 0,C 180,E1 10652.48,E2 10652.48} C_VEL
LIN {X 0,Y 247.59,Z 922.393,A -85,B 0,C 180,E1 10647.673,E2 10647.673} C_VEL
LIN {X 0,Y 237.26,Z 922.254,A -85,B 0,C 180,E1 10642.551,E2 10642.551} C_VEL
LIN {X 0,Y 229.826,Z 920.318,A -85,B 0,C 180,E1 10637.469,E2 10637.469} C_VEL
LIN {X 0,Y 224.59,Z 916.719,A -85,B 0,C 180,E1 10632.339,E2 10632.339} C_VEL
LIN {X 0,Y 221.083,Z 911.282,A -85,B 0,C 180,E1 10627.014,E2 10627.014} C_VEL
LIN {X 0,Y 219.198,Z 904.22,A -85,B 0,C 180,E1 10621.83,E2 10621.83} C_VEL
LIN {X 0,Y 218.489,Z 896.148,A -85,B 0,C 180,E1 10617.114,E2 10617.114} C_VEL
LIN {X 0,Y 218.603,Z 886.203,A -85,B 0,C 180,E1 10612.377,E2 10612.377} C_VEL
LIN {X 0,Y 219.538,Z 874.118,A -85,B 0,C 180,E1 10607.639,E2 10607.639} C_VEL
LIN {X 0,Y 221.278,Z 860.483,A -85,B 0,C 180,E1 10603.19,E2 10603.19} C_VEL
LIN {X 0,Y 223.838,Z 844.818,A -85,B 0,C 180,E1 10598.925,E2 10598.925} C_VEL
LIN {X 0,Y 227.068,Z 827.49,A -85,B 0,C 180,E1 10594.992,E2 10594.992} C_VEL
LIN {X 0,Y 227.792,Z 823.98,A -85,B 0,C 180,E1 10594.243,E2 10594.243} C_VEL
LIN {X 0,Y 229.332,Z 823.711,A -85,B 0,C 180,E1 10593.315,E2 10593.315} C_VEL
LIN {X 0,Y 232.306,Z 822.132,A -85,B 0,C 180,E1 10592.299,E2 10592.299} C_VEL
LIN {X 0,Y 233.62,Z 821.352,A -85,B 0,C 180,E1 10591.914,E2 10591.914} C_VEL
LIN {X 0,Y 236.802,Z 820.097,A -85,B 0,C 180,E1 10590.672,E2 10590.672} C_VEL
LIN {X 0,Y 240.216,Z 818.14,A -85,B 0,C 180,E1 10589.757,E2 10589.757} C_VEL
LIN {X 0,Y 244.439,Z 816.324,A -85,B 0,C 180,E1 10588.426,E2 10588.426} C_VEL
LIN {X 0,Y 248.707,Z 813.984,A -85,B 0,C 180,E1 10587.403,E2 10587.403} C_VEL
LIN {X 0,Y 254.451,Z 811.105,A -85,B 0,C 180,E1 10586.012,E2 10586.012} C_VEL
LIN {X 0,Y 258.017,Z 809.132,A -85,B 0,C 180,E1 10585.273,E2 10585.273} C_VEL
LIN {X 0,Y 263.968,Z 805.958,A -85,B 0,C 180,E1 10584.046,E2 10584.046} C_VEL
LIN {X 0,Y 268.061,Z 803.474,A -85,B 0,C 180,E1 10583.358,E2 10583.358} C_VEL
LIN {X 0,Y 275.267,Z 799.382,A -85,B 0,C 180,E1 10582.129,E2 10582.129} C_VEL
LIN {X 0,Y 280.509,Z 796.003,A -85,B 0,C 180,E1 10581.406,E2 10581.406} C_VEL
LIN {X 0,Y 285.552,Z 793.118,A -85,B 0,C 180,E1 10580.63,E2 10580.63} C_VEL
LIN {X 0,Y 277.304,Z 810.392,A -85,B 0,C 180,E1 10578.159,E2 10578.159} C_VEL
LIN {X 0,Y 268.686,Z 826.509,A -85,B 0,C 180,E1 10575.299,E2 10575.299} C_VEL
LIN {X 0,Y 259.94,Z 841.364,A -85,B 0,C 180,E1 10572.014,E2 10572.014} C_VEL
LIN {X 0,Y 251.484,Z 854.656,A -85,B 0,C 180,E1 10568.335,E2 10568.335} C_VEL
LIN {X 0,Y 243.538,Z 866.423,A -85,B 0,C 180,E1 10564.228,E2 10564.228} C_VEL
LIN {X 0,Y 236.357,Z 876.652,A -85,B 0,C 180,E1 10559.667,E2 10559.667} C_VEL
LIN {X 0,Y 230.446,Z 884.952,A -85,B 0,C 180,E1 10554.89,E2 10554.89} C_VEL
LIN {X 0,Y 225.652,Z 891.77,A -85,B 0,C 180,E1 10549.68,E2 10549.68} C_VEL
LIN {X 0,Y 222.258,Z 896.813,A -85,B 0,C 180,E1 10544.326,E2 10544.326} C_VEL
LIN {X 0,Y 220.105,Z 900.288,A -85,B 0,C 180,E1 10538.622,E2 10538.622} C_VEL
LIN {X 0,Y 219.163,Z 901.958,A -85,B 0,C 180,E1 10533.139,E2 10533.139} C_VEL
LIN {X 0,Y 219.078,Z 902.088,A -85,B 0,C 180,E1 10527.908,E2 10527.908} C_VEL
LIN {X 0,Y 219.828,Z 900.735,A -85,B 0,C 180,E1 10522.42,E2 10522.42} C_VEL
LIN {X 0,Y 221.607,Z 897.812,A -85,B 0,C 180,E1 10516.962,E2 10516.962} C_VEL
LIN {X 0,Y 224.89,Z 892.917,A -85,B 0,C 180,E1 10511.268,E2 10511.268} C_VEL
LIN {X 0,Y 229.595,Z 886.207,A -85,B 0,C 180,E1 10505.835,E2 10505.835} C_VEL
LIN {X 0,Y 235.615,Z 877.788,A -85,B 0,C 180,E1 10500.789,E2 10500.789} C_VEL
LIN {X 0,Y 242.277,Z 868.356,A -85,B 0,C 180,E1 10496.425,E2 10496.425} C_VEL
LIN {X 0,Y 250.04,Z 856.97,A -85,B 0,C 180,E1 10492.278,E2 10492.278} C_VEL
LIN {X 0,Y 258.343,Z 844.109,A -85,B 0,C 180,E1 10488.56,E2 10488.56} C_VEL
LIN {X 0,Y 266.959,Z 829.748,A -85,B 0,C 180,E1 10485.239,E2 10485.239} C_VEL
LIN {X 0,Y 275.684,Z 813.801,A -85,B 0,C 180,E1 10482.278,E2 10482.278} C_VEL
LIN {X 0,Y 283.965,Z 796.943,A -85,B 0,C 180,E1 10479.754,E2 10479.754} C_VEL
LIN {X 0,Y 291.586,Z 779.329,A -85,B 0,C 180,E1 10477.615,E2 10477.615} C_VEL
LIN {X 0,Y 298.391,Z 761.127,A -85,B 0,C 180,E1 10475.814,E2 10475.814} C_VEL
LIN {X 0,Y 304.38,Z 742.174,A -85,B 0,C 180,E1 10474.292,E2 10474.292} C_VEL
LIN {X 0,Y 309.449,Z 722.453,A -85,B 0,C 180,E1 10473.019,E2 10473.019} C_VEL
LIN {X 0,Y 313.937,Z 699.919,A -85,B 0,C 180,E1 10471.876,E2 10471.876} C_VEL
LIN {X 0,Y 321.08,Z 660.976,A -85,B 0,C 180,E1 10470.289,E2 10470.289} C_VEL
LIN {X 0,Y 328.367,Z 619.459,A -85,B 0,C 180,E1 10469.003,E2 10469.003} C_VEL
LIN {X 0,Y 335.529,Z 572.373,A -85,B 0,C 180,E1 10467.831,E2 10467.831} C_VEL
LIN {X 0,Y 341.072,Z 525.516,A -85,B 0,C 180,E1 10466.862,E2 10466.862} C_VEL
LIN {X 0,Y 346.043,Z 470.407,A -85,B 0,C 180,E1 10465.886,E2 10465.886} C_VEL
LIN {X 0,Y 346.243,Z 465.398,A -85,B 0,C 180,E1 10465.64,E2 10465.64} C_VEL
LIN {X 0,Y 346.398,Z 453.089,A -85,B 0,C 180,E1 10464.378,E2 10464.378} C_VEL
LIN {X 0,Y 347.142,Z 448.885,A -85,B 0,C 180,E1 10464.14,E2 10464.14} C_VEL
LIN {X 0,Y 347.825,Z 446.041,A -85,B 0,C 180,E1 10464.052,E2 10464.052} C_VEL
LIN {X 0,Y 344.964,Z 434.776,A -85,B 0,C 180,E1 10461.109,E2 10461.109} C_VEL
LIN {X 0,Y 342.252,Z 424.826,A -85,B 0,C 180,E1 10457.952,E2 10457.952} C_VEL
LIN {X 0,Y 339.928,Z 416.846,A -85,B 0,C 180,E1 10454.828,E2 10454.828} C_VEL
LIN {X 0,Y 338.009,Z 410.266,A -85,B 0,C 180,E1 10451.605,E2 10451.605} C_VEL
LIN {X 0,Y 336.969,Z 406.588,A -85,B 0,C 180,E1 10449.307,E2 10449.307} C_VEL
LIN {X 0,Y 336.176,Z 403.515,A -85,B 0,C 180,E1 10447.005,E2 10447.005} C_VEL
LIN {X 0,Y 335.703,Z 399.838,A -85,B 0,C 180,E1 10443.244,E2 10443.244} C_VEL
LIN {X 0,Y 336.154,Z 398.855,A -85,B 0,C 180,E1 10437.954,E2 10437.954} C_VEL
LIN {X 0,Y 337.525,Z 399.846,A -85,B 0,C 180,E1 10434.56,E2 10434.56} C_VEL
LIN {X 0,Y 338.217,Z 411.43,A -85,B 0,C 180,E1 10430.642,E2 10430.642} C_VEL
LIN {X 0,Y 339.496,Z 420.899,A -85,B 0,C 180,E1 10427.843,E2 10427.843} C_VEL
LIN {X 0,Y 342.954,Z 437.759,A -85,B 0,C 180,E1 10423.442,E2 10423.442} C_VEL
LIN {X 0,Y 343.815,Z 442.334,A -85,B 0,C 180,E1 10422.482,E2 10422.482} C_VEL
LIN {X 0,Y 324.701,Z 558.02,A -85,B 0,C 180,E1 10419.465,E2 10419.465} C_VEL
LIN {X 0,Y 319.052,Z 621.611,A -85,B 0,C 180,E1 10418.116,E2 10418.116} C_VEL
LIN {X 0,Y 314.329,Z 657.117,A -85,B 0,C 180,E1 10417.25,E2 10417.25} C_VEL
LIN {X 0,Y 308.487,Z 691.069,A -85,B 0,C 180,E1 10416.199,E2 10416.199} C_VEL
LIN {X 0,Y 301.049,Z 726.478,A -85,B 0,C 180,E1 10414.838,E2 10414.838} C_VEL
LIN {X 0,Y 293.63,Z 757.559,A -85,B 0,C 180,E1 10413.289,E2 10413.289} C_VEL
LIN {X 0,Y 285.371,Z 788.213,A -85,B 0,C 180,E1 10411.367,E2 10411.367} C_VEL
LIN {X 0,Y 279.619,Z 806.503,A -85,B 0,C 180,E1 10409.924,E2 10409.924} C_VEL
LIN {X 0,Y 272.693,Z 824.978,A -85,B 0,C 180,E1 10408.129,E2 10408.129} C_VEL
LIN {X 0,Y 264.997,Z 842.919,A -85,B 0,C 180,E1 10405.947,E2 10405.947} C_VEL
LIN {X 0,Y 256.789,Z 860.091,A -85,B 0,C 180,E1 10403.334,E2 10403.334} C_VEL
LIN {X 0,Y 248.598,Z 875.732,A -85,B 0,C 180,E1 10400.375,E2 10400.375} C_VEL
LIN {X 0,Y 240.08,Z 890.924,A -85,B 0,C 180,E1 10396.789,E2 10396.789} C_VEL
LIN {X 0,Y 232.336,Z 904.2,A -85,B 0,C 180,E1 10392.841,E2 10392.841} C_VEL
LIN {X 0,Y 225.293,Z 916.132,A -85,B 0,C 180,E1 10388.414,E2 10388.414} C_VEL
LIN {X 0,Y 219.007,Z 927.216,A -85,B 0,C 180,E1 10383.221,E2 10383.221} C_VEL
LIN {X 0,Y 214.367,Z 936.293,A -85,B 0,C 180,E1 10377.803,E2 10377.803} C_VEL
LIN {X 0,Y 211.27,Z 943.925,A -85,B 0,C 180,E1 10371.932,E2 10371.932} C_VEL
LIN {X 0,Y 209.887,Z 949.622,A -85,B 0,C 180,E1 10366.04,E2 10366.04} C_VEL
LIN {X 0,Y 209.829,Z 953.456,A -85,B 0,C 180,E1 10360.433,E2 10360.433} C_VEL
LIN {X 0,Y 210.451,Z 955.606,A -85,B 0,C 180,E1 10355.453,E2 10355.453} C_VEL
LIN {X 0,Y 210.953,Z 956.378,A -85,B 0,C 180,E1 10351.086,E2 10351.086} C_VEL
LIN {X 0,Y 210.827,Z 956.176,A -85,B 0,C 180,E1 10347.009,E2 10347.009} C_VEL
LIN {X 0,Y 210.324,Z 955.42,A -85,B 0,C 180,E1 10343.174,E2 10343.174} C_VEL
LIN {X 0,Y 209.602,Z 955.36,A -85,B 0,C 180,E1 10337.604,E2 10337.604} C_VEL
LIN {X 0,Y 210.22,Z 953.841,A -85,B 0,C 180,E1 10330.841,E2 10330.841} C_VEL
LIN {X 0,Y 214.082,Z 950.092,A -85,B 0,C 180,E1 10322.76,E2 10322.76} C_VEL
LIN {X 0,Y 222.093,Z 944.496,A -85,B 0,C 180,E1 10314.811,E2 10314.811} C_VEL
LIN {X 0,Y 235.722,Z 936.412,A -85,B 0,C 180,E1 10306.853,E2 10306.853} C_VEL
LIN {X 0,Y 254.87,Z 926.374,A -85,B 0,C 180,E1 10299.741,E2 10299.741} C_VEL
LIN {X 0,Y 266.015,Z 920.808,A -85,B 0,C 180,E1 10296.702,E2 10296.702} C_VEL
LIN {X 0,Y 250.517,Z 923.428,A -85,B 0,C 180,E1 10292.204,E2 10292.204} C_VEL
LIN {X 0,Y 237.812,Z 924.193,A -85,B 0,C 180,E1 10287.277,E2 10287.277} C_VEL
LIN {X 0,Y 228.43,Z 923.252,A -85,B 0,C 180,E1 10282.385,E2 10282.385} C_VEL
LIN {X 0,Y 221.072,Z 920.618,A -85,B 0,C 180,E1 10277.097,E2 10277.097} C_VEL
LIN {X 0,Y 215.973,Z 916.354,A -85,B 0,C 180,E1 10271.754,E2 10271.754} C_VEL
LIN {X 0,Y 212.767,Z 910.583,A -85,B 0,C 180,E1 10266.476,E2 10266.476} C_VEL
LIN {X 0,Y 211.014,Z 902.853,A -85,B 0,C 180,E1 10261.056,E2 10261.056} C_VEL
LIN {X 0,Y 210.442,Z 893.66,A -85,B 0,C 180,E1 10255.913,E2 10255.913} C_VEL
LIN {X 0,Y 210.785,Z 882.923,A -85,B 0,C 180,E1 10250.994,E2 10250.994} C_VEL
LIN {X 0,Y 211.915,Z 870.762,A -85,B 0,C 180,E1 10246.354,E2 10246.354} C_VEL
LIN {X 0,Y 213.952,Z 856.352,A -85,B 0,C 180,E1 10241.753,E2 10241.753} C_VEL
LIN {X 0,Y 216.755,Z 840.361,A -85,B 0,C 180,E1 10237.488,E2 10237.488} C_VEL
LIN {X 0,Y 218.378,Z 832.199,A -85,B 0,C 180,E1 10235.52,E2 10235.52} C_VEL
LIN {X 0,Y 220.054,Z 831.839,A -85,B 0,C 180,E1 10234.427,E2 10234.427} C_VEL
LIN {X 0,Y 223.639,Z 829.907,A -85,B 0,C 180,E1 10233.155,E2 10233.155} C_VEL
LIN {X 0,Y 226.592,Z 828.838,A -85,B 0,C 180,E1 10231.825,E2 10231.825} C_VEL
LIN {X 0,Y 230.34,Z 826.932,A -85,B 0,C 180,E1 10230.625,E2 10230.625} C_VEL
LIN {X 0,Y 234.504,Z 825.124,A -85,B 0,C 180,E1 10229.225,E2 10229.225} C_VEL
LIN {X 0,Y 237.283,Z 823.677,A -85,B 0,C 180,E1 10228.498,E2 10228.498} C_VEL
LIN {X 0,Y 242.468,Z 821.37,A -85,B 0,C 180,E1 10227.02,E2 10227.02} C_VEL
LIN {X 0,Y 246.111,Z 819.479,A -85,B 0,C 180,E1 10226.179,E2 10226.179} C_VEL
LIN {X 0,Y 252.074,Z 816.571,A -85,B 0,C 180,E1 10224.799,E2 10224.799} C_VEL
LIN {X 0,Y 255.675,Z 814.634,A -85,B 0,C 180,E1 10224.082,E2 10224.082} C_VEL
LIN {X 0,Y 262.61,Z 811.083,A -85,B 0,C 180,E1 10222.742,E2 10222.742} C_VEL
LIN {X 0,Y 267.555,Z 808.331,A -85,B 0,C 180,E1 10221.929,E2 10221.929} C_VEL
LIN {X 0,Y 275.109,Z 804.086,A -85,B 0,C 180,E1 10220.772,E2 10220.772} C_VEL
LIN {X 0,Y 276.135,Z 803.504,A -85,B 0,C 180,E1 10220.618,E2 10220.618} C_VEL
LIN {X 0,Y 267.372,Z 820.191,A -85,B 0,C 180,E1 10217.931,E2 10217.931} C_VEL
LIN {X 0,Y 258.262,Z 835.758,A -85,B 0,C 180,E1 10214.8,E2 10214.8} C_VEL
LIN {X 0,Y 249.569,Z 849.375,A -85,B 0,C 180,E1 10211.382,E2 10211.382} C_VEL
LIN {X 0,Y 240.778,Z 862.18,A -85,B 0,C 180,E1 10207.323,E2 10207.323} C_VEL
LIN {X 0,Y 233.059,Z 872.853,A -85,B 0,C 180,E1 10203.016,E2 10203.016} C_VEL
LIN {X 0,Y 226.167,Z 882.078,A -85,B 0,C 180,E1 10198.233,E2 10198.233} C_VEL
LIN {X 0,Y 220.376,Z 889.781,A -85,B 0,C 180,E1 10192.967,E2 10192.967} C_VEL
LIN {X 0,Y 216.078,Z 895.64,A -85,B 0,C 180,E1 10187.505,E2 10187.505} C_VEL
LIN {X 0,Y 213.212,Z 899.787,A -85,B 0,C 180,E1 10181.908,E2 10181.908} C_VEL
LIN {X 0,Y 211.636,Z 902.278,A -85,B 0,C 180,E1 10176.239,E2 10176.239} C_VEL
LIN {X 0,Y 211.092,Z 903.177,A -85,B 0,C 180,E1 10170.814,E2 10170.814} C_VEL
LIN {X 0,Y 211.364,Z 902.697,A -85,B 0,C 180,E1 10165.387,E2 10165.387} C_VEL
LIN {X 0,Y 212.614,Z 900.69,A -85,B 0,C 180,E1 10159.706,E2 10159.706} C_VEL
LIN {X 0,Y 215.071,Z 897.086,A -85,B 0,C 180,E1 10154.08,E2 10154.08} C_VEL
LIN {X 0,Y 218.936,Z 891.789,A -85,B 0,C 180,E1 10148.57,E2 10148.57} C_VEL
LIN {X 0,Y 224,Z 885.074,A -85,B 0,C 180,E1 10143.488,E2 10143.488} C_VEL
LIN {X 0,Y 230.407,Z 876.576,A -85,B 0,C 180,E1 10138.617,E2 10138.617} C_VEL
LIN {X 0,Y 238.113,Z 866.087,A -85,B 0,C 180,E1 10133.993,E2 10133.993} C_VEL
LIN {X 0,Y 246.102,Z 854.75,A -85,B 0,C 180,E1 10130.063,E2 10130.063} C_VEL
LIN {X 0,Y 254.985,Z 841.256,A -85,B 0,C 180,E1 10126.357,E2 10126.357} C_VEL
LIN {X 0,Y 263.722,Z 826.902,A -85,B 0,C 180,E1 10123.204,E2 10123.204} C_VEL
LIN {X 0,Y 272.5,Z 810.986,A -85,B 0,C 180,E1 10120.391,E2 10120.391} C_VEL
LIN {X 0,Y 280.898,Z 793.934,A -85,B 0,C 180,E1 10117.959,E2 10117.959} C_VEL
LIN {X 0,Y 288.397,Z 776.609,A -85,B 0,C 180,E1 10115.947,E2 10115.947} C_VEL
LIN {X 0,Y 295.434,Z 757.617,A -85,B 0,C 180,E1 10114.157,E2 10114.157} C_VEL
LIN {X 0,Y 301.413,Z 738.331,A -85,B 0,C 180,E1 10112.695,E2 10112.695} C_VEL
LIN {X 0,Y 306.434,Z 718.043,A -85,B 0,C 180,E1 10111.466,E2 10111.466} C_VEL
LIN {X 0,Y 313.749,Z 680.473,A -85,B 0,C 180,E1 10109.746,E2 10109.746} C_VEL
LIN {X 0,Y 321.162,Z 640.371,A -85,B 0,C 180,E1 10108.333,E2 10108.333} C_VEL
LIN {X 0,Y 328.989,Z 593.753,A -85,B 0,C 180,E1 10107.087,E2 10107.087} C_VEL
LIN {X 0,Y 335.28,Z 547.106,A -85,B 0,C 180,E1 10106.057,E2 10106.057} C_VEL
LIN {X 0,Y 340.536,Z 494.772,A -85,B 0,C 180,E1 10105.09,E2 10105.09} C_VEL
LIN {X 0,Y 343.544,Z 463.899,A -85,B 0,C 180,E1 10104.546,E2 10104.546} C_VEL
LIN {X 0,Y 347.142,Z 448.885,A -85,B 0,C 180,E1 10104.14,E2 10104.14} C_VEL
LIN {X 0,Y 347.548,Z 445.802,A -85,B 0,C 180,E1 10103.894,E2 10103.894} C_VEL
LIN {X 0,Y 347.187,Z 442.834,A -85,B 0,C 180,E1 10103.322,E2 10103.322} C_VEL
LIN {X 0,Y 345.794,Z 440.355,A -85,B 0,C 180,E1 10102.334,E2 10102.334} C_VEL
LIN {X 0,Y 341.285,Z 437.262,A -85,B 0,C 180,E1 10099.503,E2 10099.503} C_VEL
LIN {X 0,Y 340.469,Z 435.442,A -85,B 0,C 180,E1 10098.706,E2 10098.706} C_VEL
LIN {X 0,Y 338.282,Z 427.186,A -85,B 0,C 180,E1 10095.735,E2 10095.735} C_VEL
LIN {X 0,Y 336.371,Z 420.098,A -85,B 0,C 180,E1 10092.533,E2 10092.533} C_VEL
LIN {X 0,Y 335.021,Z 414.87,A -85,B 0,C 180,E1 10089.621,E2 10089.621} C_VEL
LIN {X 0,Y 334.091,Z 411.077,A -85,B 0,C 180,E1 10086.703,E2 10086.703} C_VEL
LIN {X 0,Y 333.789,Z 407.578,A -85,B 0,C 180,E1 10083.091,E2 10083.091} C_VEL
LIN {X 0,Y 334.325,Z 406.643,A -85,B 0,C 180,E1 10077.943,E2 10077.943} C_VEL
LIN {X 0,Y 335.554,Z 407.569,A -85,B 0,C 180,E1 10074.871,E2 10074.871} C_VEL
LIN {X 0,Y 336.427,Z 420.93,A -85,B 0,C 180,E1 10070.376,E2 10070.376} C_VEL
LIN {X 0,Y 339.49,Z 440.436,A -85,B 0,C 180,E1 10065.027,E2 10065.027} C_VEL
LIN {X 0,Y 340.649,Z 446.205,A -85,B 0,C 180,E1 10063.666,E2 10063.666} C_VEL
LIN {X 0,Y 322.123,Z 555.167,A -85,B 0,C 180,E1 10060.857,E2 10060.857} C_VEL
LIN {X 0,Y 316.245,Z 619.304,A -85,B 0,C 180,E1 10059.5,E2 10059.5} C_VEL
LIN {X 0,Y 311.347,Z 655.198,A -85,B 0,C 180,E1 10058.643,E2 10058.643} C_VEL
LIN {X 0,Y 305.407,Z 688.827,A -85,B 0,C 180,E1 10057.621,E2 10057.621} C_VEL
LIN {X 0,Y 297.92,Z 723.828,A -85,B 0,C 180,E1 10056.309,E2 10056.309} C_VEL
LIN {X 0,Y 290.514,Z 754.277,A -85,B 0,C 180,E1 10054.849,E2 10054.849} C_VEL
LIN {X 0,Y 281.87,Z 785.806,A -85,B 0,C 180,E1 10052.921,E2 10052.921} C_VEL
LIN {X 0,Y 275.545,Z 805.229,A -85,B 0,C 180,E1 10051.421,E2 10051.421} C_VEL
LIN {X 0,Y 267.973,Z 824.701,A -85,B 0,C 180,E1 10049.534,E2 10049.534} C_VEL
LIN {X 0,Y 260.035,Z 842.471,A -85,B 0,C 180,E1 10047.363,E2 10047.363} C_VEL
LIN {X 0,Y 251.6,Z 859.39,A -85,B 0,C 180,E1 10044.774,E2 10044.774} C_VEL
LIN {X 0,Y 242.748,Z 875.525,A -85,B 0,C 180,E1 10041.691,E2 10041.691} C_VEL
LIN {X 0,Y 233.873,Z 890.528,A -85,B 0,C 180,E1 10038.065,E2 10038.065} C_VEL
LIN {X 0,Y 225.322,Z 904.412,A -85,B 0,C 180,E1 10033.81,E2 10033.81} C_VEL
LIN {X 0,Y 217.625,Z 916.766,A -85,B 0,C 180,E1 10029.01,E2 10029.01} C_VEL
LIN {X 0,Y 211.432,Z 927.087,A -85,B 0,C 180,E1 10023.92,E2 10023.92} C_VEL
LIN {X 0,Y 206.508,Z 936.172,A -85,B 0,C 180,E1 10018.209,E2 10018.209} C_VEL
LIN {X 0,Y 203.356,Z 943.418,A -85,B 0,C 180,E1 10012.247,E2 10012.247} C_VEL
LIN {X 0,Y 201.913,Z 948.996,A -85,B 0,C 180,E1 10006.1,E2 10006.1} C_VEL
LIN {X 0,Y 201.905,Z 952.845,A -85,B 0,C 180,E1 9999.981,E2 9999.981} C_VEL
LIN {X 0,Y 202.637,Z 954.84,A -85,B 0,C 180,E1 9994.62,E2 9994.62} C_VEL
LIN {X 0,Y 203.037,Z 955.434,A -85,B 0,C 180,E1 9990.282,E2 9990.282} C_VEL
LIN {X 0,Y 202.771,Z 954.989,A -85,B 0,C 180,E1 9986.041,E2 9986.041} C_VEL
LIN {X 0,Y 202.19,Z 953.885,A -85,B 0,C 180,E1 9981.468,E2 9981.468} C_VEL
LIN {X 0,Y 201.691,Z 953.677,A -85,B 0,C 180,E1 9975.648,E2 9975.648} C_VEL
LIN {X 0,Y 202.951,Z 952.051,A -85,B 0,C 180,E1 9968.616,E2 9968.616} C_VEL
LIN {X 0,Y 208.335,Z 947.988,A -85,B 0,C 180,E1 9959.739,E2 9959.739} C_VEL
LIN {X 0,Y 218.347,Z 942.174,A -85,B 0,C 180,E1 9951.479,E2 9951.479} C_VEL
LIN {X 0,Y 234.358,Z 934.019,A -85,B 0,C 180,E1 9943.505,E2 9943.505} C_VEL
LIN {X 0,Y 254.283,Z 924.78,A -85,B 0,C 180,E1 9937.038,E2 9937.038} C_VEL
LIN {X 0,Y 255.683,Z 924.14,A -85,B 0,C 180,E1 9936.611,E2 9936.611} C_VEL
LIN {X 0,Y 240.072,Z 925.76,A -85,B 0,C 180,E1 9931.826,E2 9931.826} C_VEL
LIN {X 0,Y 228.015,Z 925.552,A -85,B 0,C 180,E1 9926.851,E2 9926.851} C_VEL
LIN {X 0,Y 218.832,Z 923.767,A -85,B 0,C 180,E1 9921.722,E2 9921.722} C_VEL
LIN {X 0,Y 212.032,Z 920.47,A -85,B 0,C 180,E1 9916.436,E2 9916.436} C_VEL
LIN {X 0,Y 207.169,Z 915.443,A -85,B 0,C 180,E1 9910.85,E2 9910.85} C_VEL
LIN {X 0,Y 204.129,Z 908.473,A -85,B 0,C 180,E1 9905.058,E2 9905.058} C_VEL
LIN {X 0,Y 202.762,Z 900.32,A -85,B 0,C 180,E1 9899.717,E2 9899.717} C_VEL
LIN {X 0,Y 202.452,Z 890.814,A -85,B 0,C 180,E1 9894.615,E2 9894.615} C_VEL
LIN {X 0,Y 203.044,Z 879.3,A -85,B 0,C 180,E1 9889.502,E2 9889.502} C_VEL
LIN {X 0,Y 204.494,Z 866.311,A -85,B 0,C 180,E1 9884.69,E2 9884.69} C_VEL
LIN {X 0,Y 206.922,Z 850.934,A -85,B 0,C 180,E1 9879.935,E2 9879.935} C_VEL
LIN {X 0,Y 208.98,Z 840.037,A -85,B 0,C 180,E1 9876.974,E2 9876.974} C_VEL
LIN {X 0,Y 210.871,Z 839.52,A -85,B 0,C 180,E1 9875.636,E2 9875.636} C_VEL
